SPLINE
SPL {X  -162.485, Y  +370.062, Z    +0.000, E1   +10.606, E3 +565885.380}
SPL {X  -162.818, Y  +379.636, Z    +0.000, E1    +5.115, E3 +565874.729}
SPL {X  -162.820, Y  +386.976, Z    +0.000, E1    +0.144, E3 +565873.828}
SPL {X  -162.820, Y  +391.982, Z    +0.000, E1    -3.443, E3 +565880.593}
SPL {X  -162.820, Y  +399.630, Z    +0.000, E1    -9.426, E3 +565883.100}
SPL {X  -162.820, Y  +408.127, Z    +0.000, E1   -18.417, E3 +565869.388}
SPL {X  -162.820, Y  +420.083, Z    +0.000, E1   -24.325, E3 +565889.864}
SPL {X  -162.820, Y  +428.527, Z    +0.000, E1   -26.988, E3 +565907.156}
SPL {X  -162.820, Y  +431.336, Z    +0.000, E1   -24.162, E3 +565937.366}
SPL {X  -162.820, Y  +432.048, Z    +0.000, E1   -22.832, E3 +565951.870}
SPL {X  -162.820, Y  +434.888, Z    +0.000, E1   -22.823, E3 +565965.819}
SPL {X  -162.820, Y  +436.834, Z    +0.000, E1   -22.779, E3 +565975.779}
SPL {X  -162.820, Y  +438.868, Z    +0.000, E1   -22.837, E3 +565985.433}
SPL {X  -162.820, Y  +441.351, Z    +0.000, E1   -22.805, E3 +565998.008}
SPL {X  -162.820, Y  +443.809, Z    +0.000, E1   -22.804, E3 +566010.174}
SPL {X  -162.820, Y  +446.105, Z    +0.000, E1   -22.815, E3 +566021.417}
SPL {X  -162.820, Y  +447.974, Z    +0.000, E1   -22.856, E3 +566030.320}
SPL {X  -162.820, Y  +449.911, Z    +0.000, E1   -22.774, E3 +566040.594}
SPL {X  -162.820, Y  +451.861, Z    +0.000, E1   -22.750, E3 +566050.442}
SPL {X  -162.820, Y  +454.167, Z    +0.000, E1   -22.842, E3 +566061.171}
SPL {X  -162.820, Y  +456.529, Z    +0.000, E1   -22.855, E3 +566072.700}
SPL {X  -162.820, Y  +458.725, Z    +0.000, E1   -22.793, E3 +566084.104}
SPL {X  -162.820, Y  +460.754, Z    +0.000, E1   -22.806, E3 +566093.977}
SPL {X  -162.820, Y  +462.409, Z    +0.000, E1   -22.783, E3 +566102.394}
SPL {X  -162.820, Y  +464.633, Z    +0.000, E1   -22.813, E3 +566113.223}
SPL {X  -162.820, Y  +467.913, Z    +0.000, E1   -22.879, E3 +566129.062}
SPL {X  -162.820, Y  +470.892, Z    +0.000, E1   -22.837, E3 +566143.952}
SPL {X  -162.820, Y  +472.726, Z    +0.000, E1   -22.777, E3 +566153.490}
SPL {X  -162.820, Y  +475.118, Z    +0.000, E1   -22.777, E3 +566165.462}
SPL {X  -162.820, Y  +478.177, Z    +0.000, E1   -22.834, E3 +566180.155}
SPL {X  -162.820, Y  +481.034, Z    +0.000, E1   -22.831, E3 +566194.292}
SPL {X  -162.820, Y  +483.391, Z    +0.000, E1   -22.793, E3 +566206.228}
SPL {X  -162.820, Y  +486.307, Z    +0.000, E1   -22.833, E3 +566220.482}
SPL {X  -162.820, Y  +488.828, Z    +0.000, E1   -22.793, E3 +566233.125}
SPL {X  -162.820, Y  +491.768, Z    +0.000, E1   -22.852, E3 +566247.422}
SPL {X  -162.820, Y  +495.526, Z    +0.000, E1   -22.833, E3 +566266.193}
SPL {X  -162.820, Y  +499.330, Z    +0.000, E1   -22.841, E3 +566284.974}
SPL {X  -162.820, Y  +503.049, Z    +0.000, E1   -22.823, E3 +566303.524}
SPL {X  -162.820, Y  +506.908, Z    +0.000, E1   -22.877, E3 +566322.194}
SPL {X  -162.820, Y  +510.068, Z    +0.000, E1   -22.761, E3 +566338.665}
SPL {X  -162.820, Y  +512.359, Z    +0.000, E1   -22.823, E3 +566349.397}
SPL {X  -162.820, Y  +513.873, Z    +0.000, E1   -22.800, E3 +566357.083}
SPL {X  -162.820, Y  +516.100, Z    +0.000, E1   -22.809, E3 +566368.160}
SPL {X  -162.820, Y  +518.662, Z    +0.000, E1   -22.847, E3 +566380.459}
SPL {X  -162.820, Y  +520.641, Z    +0.000, E1   -22.790, E3 +566390.699}
SPL {X  -162.820, Y  +523.535, Z    +0.000, E1   -22.857, E3 +566404.668}
SPL {X  -162.820, Y  +526.661, Z    +0.000, E1   -22.801, E3 +566420.492}
SPL {X  -162.820, Y  +528.725, Z    +0.000, E1   -22.770, E3 +566430.862}
SPL {X  -162.820, Y  +530.303, Z    +0.000, E1   -22.798, E3 +566438.481}
SPL {X  -162.820, Y  +532.614, Z    +0.000, E1   -22.828, E3 +566449.749}
SPL {X  -162.820, Y  +534.838, Z    +0.000, E1   -22.864, E3 +566460.378}
SPL {X  -162.820, Y  +536.882, Z    +0.000, E1   -22.782, E3 +566471.233}
SPL {X  -162.820, Y  +539.194, Z    +0.000, E1   -22.826, E3 +566482.282}
SPL {X  -162.820, Y  +541.555, Z    +0.000, E1   -22.817, E3 +566494.096}
SPL {X  -162.820, Y  +543.728, Z    +0.000, E1   -22.799, E3 +566504.954}
SPL {X  -162.820, Y  +545.925, Z    +0.000, E1   -22.803, E3 +566515.823}
SPL {X  -162.820, Y  +548.328, Z    +0.000, E1   -22.796, E3 +566527.819}
SPL {X  -162.820, Y  +551.027, Z    +0.000, E1   -22.819, E3 +566541.012}
SPL {X  -162.820, Y  +553.721, Z    +0.000, E1   -22.807, E3 +566554.456}
SPL {X  -162.820, Y  +556.430, Z    +0.000, E1   -22.821, E3 +566567.752}
SPL {X  -162.820, Y  +559.675, Z    +0.000, E1   -22.837, E3 +566583.832}
SPL {X  -162.820, Y  +562.799, Z    +0.000, E1   -22.814, E3 +566599.338}
SPL {X  -162.820, Y  +565.170, Z    +0.000, E1   -22.801, E3 +566611.163}
SPL {X  -162.820, Y  +568.020, Z    +0.000, E1   -22.787, E3 +566625.550}
SPL {X  -162.820, Y  +570.992, Z    +0.000, E1   -22.834, E3 +566639.769}
SPL {X  -162.820, Y  +572.901, Z    +0.000, E1   -22.775, E3 +566649.638}
SPL {X  -162.820, Y  +575.638, Z    +0.000, E1   -22.855, E3 +566662.747}
SPL {X  -162.820, Y  +578.553, Z    +0.000, E1   -22.801, E3 +566677.459}
SPL {X  -162.820, Y  +581.064, Z    +0.000, E1   -22.823, E3 +566689.744}
SPL {X  -162.820, Y  +583.435, Z    +0.000, E1   -22.808, E3 +566701.565}
SPL {X  -162.820, Y  +585.410, Z    +0.000, E1   -22.764, E3 +566711.701}
SPL {X  -162.820, Y  +587.676, Z    +0.000, E1   -22.853, E3 +566722.216}
SPL {X  -162.820, Y  +589.682, Z    +0.000, E1   -22.776, E3 +566732.746}
SPL {X  -162.820, Y  +591.720, Z    +0.000, E1   -22.868, E3 +566742.057}
SPL {X  -162.820, Y  +593.650, Z    +0.000, E1   -22.810, E3 +566752.126}
SPL {X  -162.820, Y  +595.830, Z    +0.000, E1   -22.828, E3 +566762.742}
SPL {X  -162.820, Y  +598.094, Z    +0.000, E1   -22.843, E3 +566773.855}
SPL {X  -162.820, Y  +600.420, Z    +0.000, E1   -22.826, E3 +566785.487}
SPL {X  -162.820, Y  +602.573, Z    +0.000, E1   -22.830, E3 +566796.072}
SPL {X  -162.820, Y  +604.828, Z    +0.000, E1   -22.784, E3 +566807.710}
SPL {X  -162.820, Y  +608.133, Z    +0.000, E1   -22.831, E3 +566823.828}
SPL {X  -162.820, Y  +611.103, Z    +0.000, E1   -22.785, E3 +566838.754}
SPL {X  -162.820, Y  +613.294, Z    +0.000, E1   -22.780, E3 +566849.627}
SPL {X  -162.820, Y  +615.356, Z    +0.000, E1   -22.799, E3 +566859.684}
SPL {X  -162.820, Y  +617.439, Z    +0.000, E1   -22.808, E3 +566869.942}
SPL {X  -162.820, Y  +619.665, Z    +0.000, E1   -22.817, E3 +566880.910}
SPL {X  -162.820, Y  +621.733, Z    +0.000, E1   -22.759, E3 +566891.634}
SPL {X  -162.820, Y  +624.076, Z    +0.000, E1   -22.774, E3 +566903.139}
SPL {X  -162.820, Y  +627.244, Z    +0.000, E1   -22.803, E3 +566918.822}
SPL {X  -162.820, Y  +630.349, Z    +0.000, E1   -22.766, E3 +566934.354}
SPL {X  -162.820, Y  +632.572, Z    +0.000, E1   -22.785, E3 +566945.160}
SPL {X  -162.820, Y  +634.507, Z    +0.000, E1   -22.784, E3 +566954.799}
SPL {X  -162.820, Y  +636.863, Z    +0.000, E1   -22.760, E3 +566966.721}
SPL {X  -162.820, Y  +640.111, Z    +0.000, E1   -22.809, E3 +566982.604}
SPL {X  -162.820, Y  +643.449, Z    +0.000, E1   -22.796, E3 +566999.122}
SPL {X  -162.820, Y  +645.630, Z    +0.000, E1   -22.795, E3 +567009.818}
SPL {X  -162.820, Y  +647.561, Z    +0.000, E1   -22.705, E3 +567020.268}
SPL {X  -162.820, Y  +651.051, Z    +0.000, E1   -22.833, E3 +567036.688}
SPL {X  -162.820, Y  +653.898, Z    +0.000, E1   -22.796, E3 +567050.874}
SPL {X  -162.820, Y  +656.161, Z    +0.000, E1   -22.812, E3 +567061.995}
SPL {X  -162.820, Y  +658.384, Z    +0.000, E1   -22.822, E3 +567072.862}
SPL {X  -162.820, Y  +660.215, Z    +0.000, E1   -22.649, E3 +567083.452}
SPL {X  -162.820, Y  +662.823, Z    +0.000, E1   -22.799, E3 +567095.160}
SPL {X  -162.820, Y  +665.862, Z    +0.000, E1   -22.864, E3 +567109.860}
SPL {X  -162.820, Y  +668.960, Z    +0.000, E1   -22.773, E3 +567125.810}
SPL {X  -162.820, Y  +671.605, Z    +0.000, E1   -22.777, E3 +567138.884}
SPL {X  -162.817, Y  +674.515, Z    +0.000, E1   -22.816, E3 +567153.081}
SPL {X  -162.773, Y  +677.428, Z    +0.000, E1   -22.762, E3 +567167.889}
SPL {X  -162.691, Y  +679.987, Z    +0.000, E1   -22.794, E3 +567180.302}
SPL {X  -162.559, Y  +682.717, Z    +0.000, E1   -22.726, E3 +567194.486}
SPL {X  -162.404, Y  +685.137, Z    +0.000, E1   -22.766, E3 +567206.008}
SPL {X  -162.229, Y  +687.364, Z    +0.000, E1   -22.685, E3 +567217.876}
SPL {X  -161.938, Y  +690.422, Z    +0.000, E1   -22.769, E3 +567232.283}
SPL {X  -161.065, Y  +697.344, Z    +0.000, E1   -25.698, E3 +567241.402}
SPL {X  -158.730, Y  +709.763, Z    +0.000, E1   -31.225, E3 +567250.075}
ENDSPLINE

SPLINE
SPL {X  -160.932, Y  +698.225, Z    +0.000, E1   -21.712, E3 +567281.185}
SPL {X  -161.691, Y  +692.643, Z    +0.000, E1   -17.369, E3 +567298.068}
SPL {X  -162.534, Y  +683.153, Z    +0.000, E1   -10.475, E3 +567323.535}
SPL {X  -162.820, Y  +667.630, Z    +0.000, E1    -0.882, E3 +567317.511}
SPL {X  -162.820, Y  +661.883, Z    +0.000, E1    +3.373, E3 +567322.954}
SPL {X  -162.820, Y  +655.163, Z    +0.000, E1    +8.702, E3 +567322.553}
SPL {X  -162.820, Y  +634.515, Z    +0.000, E1   +26.439, E3 +567314.966}
ENDSPLINE

SPLINE
SPL {X  -162.820, Y  +638.080, Z    +0.000, E1   +18.858, E3 +567344.931}
ENDSPLINE

SPLINE
SPL {X  -162.820, Y  +623.278, Z    +0.000, E1   +28.723, E3 +567346.501}
SPL {X  -162.820, Y  +618.658, Z    +0.000, E1   +26.841, E3 +567375.110}
ENDSPLINE

SPLINE
SPL {X  -162.820, Y  +623.685, Z    +0.000, E1   +22.346, E3 +567387.417}
ENDSPLINE

SPLINE
SPL {X  -162.820, Y  +621.304, Z    +0.000, E1   +22.259, E3 +567400.232}
SPL {X  -162.820, Y  +618.758, Z    +0.000, E1   +22.239, E3 +567413.383}
SPL {X  -162.820, Y  +616.062, Z    +0.000, E1   +22.275, E3 +567426.803}
SPL {X  -162.820, Y  +613.536, Z    +0.000, E1   +22.242, E3 +567439.925}
SPL {X  -162.820, Y  +611.128, Z    +0.000, E1   +22.252, E3 +567452.096}
SPL {X  -162.820, Y  +608.428, Z    +0.000, E1   +22.255, E3 +567465.879}
SPL {X  -162.820, Y  +605.984, Z    +0.000, E1   +22.221, E3 +567478.516}
SPL {X  -162.820, Y  +603.020, Z    +0.000, E1   +22.272, E3 +567493.414}
SPL {X  -162.820, Y  +599.168, Z    +0.000, E1   +22.310, E3 +567512.682}
SPL {X  -162.820, Y  +595.597, Z    +0.000, E1   +22.284, E3 +567531.018}
SPL {X  -162.820, Y  +593.320, Z    +0.000, E1   +22.199, E3 +567543.109}
SPL {X  -162.820, Y  +591.031, Z    +0.000, E1   +22.283, E3 +567554.200}
SPL {X  -162.820, Y  +588.026, Z    +0.000, E1   +22.301, E3 +567569.327}
SPL {X  -162.820, Y  +585.899, Z    +0.000, E1   +22.286, E3 +567580.129}
SPL {X  -162.820, Y  +583.204, Z    +0.000, E1   +22.278, E3 +567594.152}
SPL {X  -162.820, Y  +579.691, Z    +0.000, E1   +22.312, E3 +567611.639}
SPL {X  -162.820, Y  +577.460, Z    +0.000, E1   +22.218, E3 +567623.627}
SPL {X  -162.820, Y  +575.394, Z    +0.000, E1   +22.240, E3 +567634.052}
SPL {X  -162.820, Y  +572.645, Z    +0.000, E1   +22.246, E3 +567648.049}
SPL {X  -162.820, Y  +570.282, Z    +0.000, E1   +22.231, E3 +567660.100}
SPL {X  -162.820, Y  +567.961, Z    +0.000, E1   +22.247, E3 +567671.889}
SPL {X  -162.820, Y  +564.506, Z    +0.000, E1   +22.298, E3 +567689.203}
SPL {X  -162.820, Y  +561.620, Z    +0.000, E1   +22.191, E3 +567704.584}
SPL {X  -162.820, Y  +559.515, Z    +0.000, E1   +22.273, E3 +567714.586}
SPL {X  -162.820, Y  +556.723, Z    +0.000, E1   +22.309, E3 +567728.670}
SPL {X  -162.820, Y  +554.378, Z    +0.000, E1   +22.288, E3 +567740.515}
SPL {X  -162.820, Y  +552.787, Z    +0.000, E1   +22.213, E3 +567749.337}
SPL {X  -162.820, Y  +550.871, Z    +0.000, E1   +22.229, E3 +567758.932}
SPL {X  -162.820, Y  +548.168, Z    +0.000, E1   +22.298, E3 +567772.268}
SPL {X  -162.820, Y  +545.860, Z    +0.000, E1   +22.216, E3 +567784.525}
SPL {X  -162.820, Y  +543.558, Z    +0.000, E1   +22.285, E3 +567795.756}
SPL {X  -162.820, Y  +540.968, Z    +0.000, E1   +22.274, E3 +567809.028}
SPL {X  -162.820, Y  +537.857, Z    +0.000, E1   +22.280, E3 +567824.904}
SPL {X  -162.820, Y  +534.880, Z    +0.000, E1   +22.252, E3 +567840.172}
SPL {X  -162.820, Y  +532.896, Z    +0.000, E1   +22.234, E3 +567850.333}
SPL {X  -162.820, Y  +531.056, Z    +0.000, E1   +22.251, E3 +567859.615}
SPL {X  -162.820, Y  +528.708, Z    +0.000, E1   +22.319, E3 +567870.996}
SPL {X  -162.820, Y  +525.932, Z    +0.000, E1   +22.258, E3 +567885.753}
SPL {X  -162.820, Y  +522.524, Z    +0.000, E1   +22.326, E3 +567902.476}
SPL {X  -162.820, Y  +519.457, Z    +0.000, E1   +22.481, E3 +567916.605}
SPL {X  -162.820, Y  +506.285, Z    +0.000, E1   +28.538, E3 +567928.063}
SPL {X  -162.820, Y  +504.441, Z    +0.000, E1   +27.574, E3 +567942.406}
SPL {X  -162.820, Y  +502.813, Z    +0.000, E1   +26.013, E3 +567960.603}
SPL {X  -162.820, Y  +502.016, Z    +0.000, E1   +24.802, E3 +567972.946}
SPL {X  -162.820, Y  +501.060, Z    +0.000, E1   +24.081, E3 +567983.135}
SPL {X  -162.820, Y  +499.934, Z    +0.000, E1   +22.814, E3 +567999.004}
SPL {X  -162.820, Y  +498.303, Z    +0.000, E1   +21.749, E3 +568016.260}
SPL {X  -162.820, Y  +495.897, Z    +0.000, E1   +21.662, E3 +568029.414}
SPL {X  -162.820, Y  +493.717, Z    +0.000, E1   +21.704, E3 +568040.520}
SPL {X  -162.820, Y  +491.396, Z    +0.000, E1   +21.707, E3 +568052.644}
SPL {X  -162.820, Y  +489.485, Z    +0.000, E1   +21.661, E3 +568062.992}
SPL {X  -162.820, Y  +487.723, Z    +0.000, E1   +21.665, E3 +568072.195}
SPL {X  -162.820, Y  +485.661, Z    +0.000, E1   +21.712, E3 +568082.639}
SPL {X  -162.820, Y  +482.775, Z    +0.000, E1   +21.716, E3 +568097.891}
SPL {X  -162.820, Y  +479.894, Z    +0.000, E1   +21.695, E3 +568112.967}
SPL {X  -162.820, Y  +477.685, Z    +0.000, E1   +21.656, E3 +568124.905}
SPL {X  -162.820, Y  +475.419, Z    +0.000, E1   +21.711, E3 +568136.258}
SPL {X  -162.820, Y  +473.301, Z    +0.000, E1   +21.712, E3 +568147.355}
SPL {X  -162.820, Y  +470.965, Z    +0.000, E1   +21.700, E3 +568159.700}
SPL {X  -162.820, Y  +469.036, Z    +0.000, E1   +21.695, E3 +568169.743}
SPL {X  -162.820, Y  +467.138, Z    +0.000, E1   +21.678, E3 +568179.915}
SPL {X  -162.820, Y  +465.011, Z    +0.000, E1   +21.692, E3 +568190.898}
SPL {X  -162.820, Y  +462.669, Z    +0.000, E1   +21.752, E3 +568202.678}
SPL {X  -162.820, Y  +460.725, Z    +0.000, E1   +21.689, E3 +568213.291}
SPL {X  -162.820, Y  +458.666, Z    +0.000, E1   +21.695, E3 +568224.103}
SPL {X  -162.820, Y  +456.431, Z    +0.000, E1   +21.708, E3 +568235.632}
SPL {X  -162.820, Y  +454.628, Z    +0.000, E1   +21.674, E3 +568245.350}
SPL {X  -162.820, Y  +452.690, Z    +0.000, E1   +21.773, E3 +568254.624}
SPL {X  -162.820, Y  +450.610, Z    +0.000, E1   +21.698, E3 +568266.223}
SPL {X  -162.820, Y  +448.170, Z    +0.000, E1   +21.667, E3 +568279.244}
SPL {X  -162.820, Y  +446.246, Z    +0.000, E1   +21.696, E3 +568289.061}
SPL {X  -162.820, Y  +443.784, Z    +0.000, E1   +21.713, E3 +568301.848}
SPL {X  -162.820, Y  +440.567, Z    +0.000, E1   +21.731, E3 +568318.687}
SPL {X  -162.820, Y  +437.628, Z    +0.000, E1   +21.678, E3 +568334.351}
SPL {X  -162.820, Y  +435.262, Z    +0.000, E1   +21.727, E3 +568346.287}
SPL {X  -162.820, Y  +433.510, Z    +0.000, E1   +21.692, E3 +568355.701}
SPL {X  -162.820, Y  +431.492, Z    +0.000, E1   +21.686, E3 +568366.396}
SPL {X  -162.820, Y  +429.074, Z    +0.000, E1   +21.710, E3 +568378.848}
SPL {X  -162.820, Y  +427.020, Z    +0.000, E1   +21.674, E3 +568389.850}
SPL {X  -162.820, Y  +424.525, Z    +0.000, E1   +21.712, E3 +568402.763}
SPL {X  -162.820, Y  +421.144, Z    +0.000, E1   +21.719, E3 +568420.430}
SPL {X  -162.820, Y  +418.116, Z    +0.000, E1   +21.761, E3 +568435.761}
SPL {X  -162.820, Y  +416.127, Z    +0.000, E1   +21.715, E3 +568446.466}
SPL {X  -162.820, Y  +414.361, Z    +0.000, E1   +21.613, E3 +568456.653}
SPL {X  -162.820, Y  +411.450, Z    +0.000, E1   +21.710, E3 +568471.227}
SPL {X  -162.820, Y  +408.590, Z    +0.000, E1   +21.735, E3 +568485.852}
SPL {X  -162.820, Y  +406.238, Z    +0.000, E1   +21.697, E3 +568498.501}
SPL {X  -162.820, Y  +403.166, Z    +0.000, E1   +21.746, E3 +568514.307}
SPL {X  -162.820, Y  +400.348, Z    +0.000, E1   +21.713, E3 +568529.142}
SPL {X  -162.820, Y  +398.298, Z    +0.000, E1   +21.721, E3 +568539.757}
SPL {X  -162.820, Y  +396.371, Z    +0.000, E1   +21.713, E3 +568549.939}
SPL {X  -162.820, Y  +394.508, Z    +0.000, E1   +21.616, E3 +568560.495}
SPL {X  -162.820, Y  +391.777, Z    +0.000, E1   +21.714, E3 +568574.154}
SPL {X  -162.820, Y  +388.822, Z    +0.000, E1   +21.717, E3 +568589.474}
SPL {X  -162.820, Y  +386.818, Z    +0.000, E1   +21.679, E3 +568600.214}
SPL {X  -162.820, Y  +384.697, Z    +0.000, E1   +21.693, E3 +568611.284}
SPL {X  -162.820, Y  +382.288, Z    +0.000, E1   +21.742, E3 +568623.407}
SPL {X  -162.817, Y  +379.520, Z    +0.000, E1   +21.723, E3 +568638.245}
SPL {X  -162.776, Y  +376.710, Z    +0.000, E1   +21.698, E3 +568652.984}
SPL {X  -162.707, Y  +374.438, Z    +0.000, E1   +21.688, E3 +568664.988}
SPL {X  -162.607, Y  +372.171, Z    +0.000, E1   +21.692, E3 +568676.788}
SPL {X  -162.494, Y  +370.197, Z    +0.000, E1   +21.655, E3 +568687.414}
SPL {X  -162.349, Y  +368.131, Z    +0.000, E1   +21.624, E3 +568698.532}
SPL {X  -162.161, Y  +365.866, Z    +0.000, E1   +21.642, E3 +568710.217}
SPL {X  -161.651, Y  +361.024, Z    +0.000, E1   +22.970, E3 +568723.640}
SPL {X  -160.281, Y  +351.857, Z    +0.000, E1   +24.243, E3 +568758.979}
ENDSPLINE

SPLINE
SPL {X  -161.833, Y  +362.603, Z    +0.000, E1   +17.021, E3 +568773.675}
ENDSPLINE

SPLINE
SPL {X  -160.786, Y  +354.842, Z    +0.000, E1   +19.274, E3 +568805.831}
ENDSPLINE

SPLINE
SPL {X  -162.485, Y  +370.062, Z    +0.000, E1   +10.606, E3 +568812.209}
SPL {X  -162.818, Y  +379.636, Z    +0.000, E1    +5.115, E3 +568801.558}
SPL {X  -162.820, Y  +386.976, Z    +0.000, E1    +0.144, E3 +568800.657}
SPL {X  -162.820, Y  +391.982, Z    +0.000, E1    -3.443, E3 +568807.422}
SPL {X  -162.820, Y  +399.630, Z    +0.000, E1    -9.426, E3 +568809.929}
SPL {X  -162.820, Y  +408.127, Z    +0.000, E1   -18.417, E3 +568796.218}
SPL {X  -162.820, Y  +420.083, Z    +0.000, E1   -24.325, E3 +568816.693}
SPL {X  -162.820, Y  +428.527, Z    +0.000, E1   -26.988, E3 +568833.985}
SPL {X  -162.820, Y  +431.336, Z    +0.000, E1   -24.162, E3 +568864.195}
SPL {X  -162.820, Y  +432.048, Z    +0.000, E1   -22.832, E3 +568878.699}
SPL {X  -162.820, Y  +434.888, Z    +0.000, E1   -22.823, E3 +568892.648}
SPL {X  -162.820, Y  +436.834, Z    +0.000, E1   -22.779, E3 +568902.609}
SPL {X  -162.820, Y  +438.868, Z    +0.000, E1   -22.837, E3 +568912.262}
SPL {X  -162.820, Y  +441.351, Z    +0.000, E1   -22.805, E3 +568924.837}
SPL {X  -162.820, Y  +443.809, Z    +0.000, E1   -22.804, E3 +568937.004}
SPL {X  -162.820, Y  +446.105, Z    +0.000, E1   -22.815, E3 +568948.246}
SPL {X  -162.820, Y  +447.974, Z    +0.000, E1   -22.856, E3 +568957.149}
SPL {X  -162.820, Y  +449.911, Z    +0.000, E1   -22.774, E3 +568967.424}
SPL {X  -162.820, Y  +451.861, Z    +0.000, E1   -22.750, E3 +568977.271}
SPL {X  -162.820, Y  +454.167, Z    +0.000, E1   -22.842, E3 +568988.001}
SPL {X  -162.820, Y  +456.529, Z    +0.000, E1   -22.855, E3 +568999.529}
SPL {X  -162.820, Y  +458.725, Z    +0.000, E1   -22.793, E3 +569010.933}
SPL {X  -162.820, Y  +460.754, Z    +0.000, E1   -22.806, E3 +569020.806}
SPL {X  -162.820, Y  +462.409, Z    +0.000, E1   -22.783, E3 +569029.223}
SPL {X  -162.820, Y  +464.633, Z    +0.000, E1   -22.813, E3 +569040.053}
SPL {X  -162.820, Y  +467.913, Z    +0.000, E1   -22.879, E3 +569055.892}
SPL {X  -162.820, Y  +470.892, Z    +0.000, E1   -22.837, E3 +569070.781}
SPL {X  -162.820, Y  +472.726, Z    +0.000, E1   -22.777, E3 +569080.320}
SPL {X  -162.820, Y  +475.118, Z    +0.000, E1   -22.777, E3 +569092.291}
SPL {X  -162.820, Y  +477.389, Z    +0.000, E1   -22.803, E3 +569103.208}
SPL {X  -162.820, Y  +478.914, Z    +0.000, E1   -22.821, E3 +569110.599}
SPL {X  -162.820, Y  +481.034, Z    +0.000, E1   -22.831, E3 +569121.122}
SPL {X  -162.820, Y  +484.256, Z    +0.000, E1   -22.840, E3 +569137.140}
SPL {X  -162.820, Y  +487.952, Z    +0.000, E1   -22.824, E3 +569155.570}
SPL {X  -162.820, Y  +490.653, Z    +0.000, E1   -22.810, E3 +569168.840}
SPL {X  -162.820, Y  +493.233, Z    +0.000, E1   -22.844, E3 +569181.518}
SPL {X  -162.820, Y  +496.150, Z    +0.000, E1   -22.796, E3 +569196.238}
SPL {X  -162.820, Y  +498.661, Z    +0.000, E1   -22.828, E3 +569208.419}
SPL {X  -162.820, Y  +501.761, Z    +0.000, E1   -22.820, E3 +569223.987}
SPL {X  -162.820, Y  +505.323, Z    +0.000, E1   -22.838, E3 +569241.434}
SPL {X  -162.820, Y  +507.875, Z    +0.000, E1   -22.849, E3 +569253.801}
SPL {X  -162.820, Y  +510.068, Z    +0.000, E1   -22.761, E3 +569265.495}
SPL {X  -162.820, Y  +512.359, Z    +0.000, E1   -22.823, E3 +569276.226}
SPL {X  -162.820, Y  +514.562, Z    +0.000, E1   -22.806, E3 +569287.413}
SPL {X  -162.820, Y  +517.952, Z    +0.000, E1   -22.864, E3 +569303.810}
SPL {X  -162.820, Y  +520.641, Z    +0.000, E1   -22.790, E3 +569317.529}
SPL {X  -162.820, Y  +522.740, Z    +0.000, E1   -22.811, E3 +569327.771}
SPL {X  -162.820, Y  +524.628, Z    +0.000, E1   -22.846, E3 +569336.766}
SPL {X  -162.820, Y  +526.661, Z    +0.000, E1   -22.801, E3 +569347.322}
SPL {X  -162.820, Y  +529.662, Z    +0.000, E1   -22.810, E3 +569362.172}
SPL {X  -162.820, Y  +532.614, Z    +0.000, E1   -22.828, E3 +569376.579}
SPL {X  -162.820, Y  +534.838, Z    +0.000, E1   -22.864, E3 +569387.208}
SPL {X  -162.820, Y  +536.882, Z    +0.000, E1   -22.782, E3 +569398.063}
SPL {X  -162.820, Y  +539.194, Z    +0.000, E1   -22.826, E3 +569409.111}
SPL {X  -162.820, Y  +541.555, Z    +0.000, E1   -22.817, E3 +569420.925}
SPL {X  -162.820, Y  +543.728, Z    +0.000, E1   -22.799, E3 +569431.783}
SPL {X  -162.820, Y  +545.925, Z    +0.000, E1   -22.803, E3 +569442.653}
SPL {X  -162.820, Y  +548.328, Z    +0.000, E1   -22.796, E3 +569454.648}
SPL {X  -162.820, Y  +551.027, Z    +0.000, E1   -22.819, E3 +569467.841}
SPL {X  -162.820, Y  +553.721, Z    +0.000, E1   -22.807, E3 +569481.285}
SPL {X  -162.820, Y  +556.430, Z    +0.000, E1   -22.821, E3 +569494.581}
SPL {X  -162.820, Y  +558.974, Z    +0.000, E1   -22.806, E3 +569507.281}
SPL {X  -162.820, Y  +562.171, Z    +0.000, E1   -22.845, E3 +569522.979}
SPL {X  -162.820, Y  +565.170, Z    +0.000, E1   -22.801, E3 +569537.993}
SPL {X  -162.820, Y  +567.308, Z    +0.000, E1   -22.750, E3 +569549.009}
SPL {X  -162.820, Y  +570.378, Z    +0.000, E1   -22.843, E3 +569563.633}
SPL {X  -162.820, Y  +573.634, Z    +0.000, E1   -22.827, E3 +569579.776}
SPL {X  -162.820, Y  +576.228, Z    +0.000, E1   -22.814, E3 +569592.673}
SPL {X  -162.820, Y  +578.553, Z    +0.000, E1   -22.801, E3 +569604.289}
SPL {X  -162.820, Y  +581.064, Z    +0.000, E1   -22.823, E3 +569616.573}
SPL {X  -162.820, Y  +583.435, Z    +0.000, E1   -22.808, E3 +569628.395}
SPL {X  -162.820, Y  +585.410, Z    +0.000, E1   -22.764, E3 +569638.530}
SPL {X  -162.820, Y  +587.676, Z    +0.000, E1   -22.853, E3 +569649.045}
SPL {X  -162.820, Y  +590.707, Z    +0.000, E1   -22.855, E3 +569664.195}
SPL {X  -162.820, Y  +593.650, Z    +0.000, E1   -22.810, E3 +569678.956}
SPL {X  -162.820, Y  +595.830, Z    +0.000, E1   -22.828, E3 +569689.571}
SPL {X  -162.820, Y  +598.094, Z    +0.000, E1   -22.843, E3 +569700.685}
SPL {X  -162.820, Y  +600.420, Z    +0.000, E1   -22.826, E3 +569712.316}
SPL {X  -162.820, Y  +602.573, Z    +0.000, E1   -22.830, E3 +569722.901}
SPL {X  -162.820, Y  +604.828, Z    +0.000, E1   -22.784, E3 +569734.539}
SPL {X  -162.820, Y  +608.133, Z    +0.000, E1   -22.831, E3 +569750.657}
SPL {X  -162.820, Y  +611.103, Z    +0.000, E1   -22.785, E3 +569765.583}
SPL {X  -162.820, Y  +613.294, Z    +0.000, E1   -22.780, E3 +569776.456}
SPL {X  -162.820, Y  +615.356, Z    +0.000, E1   -22.799, E3 +569786.513}
SPL {X  -162.820, Y  +617.439, Z    +0.000, E1   -22.808, E3 +569796.771}
SPL {X  -162.820, Y  +619.665, Z    +0.000, E1   -22.817, E3 +569807.739}
SPL {X  -162.820, Y  +621.733, Z    +0.000, E1   -22.759, E3 +569818.464}
SPL {X  -162.820, Y  +624.076, Z    +0.000, E1   -22.774, E3 +569829.969}
SPL {X  -162.820, Y  +627.244, Z    +0.000, E1   -22.803, E3 +569845.651}
SPL {X  -162.820, Y  +630.349, Z    +0.000, E1   -22.766, E3 +569861.183}
SPL {X  -162.820, Y  +632.572, Z    +0.000, E1   -22.785, E3 +569871.989}
SPL {X  -162.820, Y  +634.507, Z    +0.000, E1   -22.784, E3 +569881.628}
SPL {X  -162.820, Y  +636.863, Z    +0.000, E1   -22.760, E3 +569893.550}
SPL {X  -162.820, Y  +640.111, Z    +0.000, E1   -22.809, E3 +569909.433}
SPL {X  -162.820, Y  +643.449, Z    +0.000, E1   -22.796, E3 +569925.951}
SPL {X  -162.820, Y  +645.630, Z    +0.000, E1   -22.795, E3 +569936.647}
SPL {X  -162.820, Y  +647.561, Z    +0.000, E1   -22.705, E3 +569947.098}
SPL {X  -162.820, Y  +651.051, Z    +0.000, E1   -22.833, E3 +569963.517}
SPL {X  -162.820, Y  +653.898, Z    +0.000, E1   -22.796, E3 +569977.703}
SPL {X  -162.820, Y  +656.161, Z    +0.000, E1   -22.812, E3 +569988.825}
SPL {X  -162.820, Y  +658.384, Z    +0.000, E1   -22.822, E3 +569999.691}
SPL {X  -162.820, Y  +660.215, Z    +0.000, E1   -22.649, E3 +570010.281}
SPL {X  -162.820, Y  +662.823, Z    +0.000, E1   -22.799, E3 +570021.989}
SPL {X  -162.820, Y  +665.112, Z    +0.000, E1   -22.835, E3 +570033.044}
SPL {X  -162.820, Y  +667.016, Z    +0.000, E1   -22.823, E3 +570042.472}
SPL {X  -162.820, Y  +668.960, Z    +0.000, E1   -22.773, E3 +570052.640}
SPL {X  -162.820, Y  +672.333, Z    +0.000, E1   -22.837, E3 +570068.976}
SPL {X  -162.812, Y  +675.071, Z    +0.000, E1   -22.742, E3 +570083.121}
SPL {X  -162.773, Y  +677.428, Z    +0.000, E1   -22.762, E3 +570094.718}
SPL {X  -162.691, Y  +679.987, Z    +0.000, E1   -22.794, E3 +570107.132}
SPL {X  -162.559, Y  +682.717, Z    +0.000, E1   -22.726, E3 +570121.315}
SPL {X  -162.349, Y  +685.880, Z    +0.000, E1   -22.738, E3 +570136.916}
SPL {X  -162.164, Y  +688.106, Z    +0.000, E1   -22.661, E3 +570148.436}
SPL {X  -161.938, Y  +690.422, Z    +0.000, E1   -22.769, E3 +570159.112}
SPL {X  -161.065, Y  +697.344, Z    +0.000, E1   -25.698, E3 +570168.231}
SPL {X  -158.553, Y  +710.529, Z    +0.000, E1   -30.890, E3 +570182.128}
ENDSPLINE

SPLINE
SPL {X  -161.215, Y  +696.305, Z    +0.000, E1   -20.575, E3 +570208.709}
SPL {X  -161.691, Y  +692.643, Z    +0.000, E1   -17.369, E3 +570224.897}
SPL {X  -162.534, Y  +683.153, Z    +0.000, E1   -10.475, E3 +570250.364}
SPL {X  -162.820, Y  +667.630, Z    +0.000, E1    -0.882, E3 +570244.340}
SPL {X  -162.820, Y  +661.883, Z    +0.000, E1    +3.373, E3 +570249.784}
SPL {X  -162.820, Y  +653.808, Z    +0.000, E1    +9.891, E3 +570247.475}
SPL {X  -162.820, Y  +632.548, Z    +0.000, E1   +27.446, E3 +570244.011}
ENDSPLINE

SPLINE
SPL {X  -162.820, Y  +638.080, Z    +0.000, E1   +18.858, E3 +570271.760}
ENDSPLINE

SPLINE
SPL {X  -162.820, Y  +623.278, Z    +0.000, E1   +28.723, E3 +570273.331}
SPL {X  -162.820, Y  +618.658, Z    +0.000, E1   +26.841, E3 +570301.939}
ENDSPLINE

SPLINE
SPL {X  -162.820, Y  +623.685, Z    +0.000, E1   +22.346, E3 +570314.246}
ENDSPLINE

SPLINE
SPL {X  -162.820, Y  +621.304, Z    +0.000, E1   +22.259, E3 +570327.061}
SPL {X  -162.820, Y  +618.758, Z    +0.000, E1   +22.239, E3 +570340.212}
SPL {X  -162.820, Y  +616.062, Z    +0.000, E1   +22.275, E3 +570353.633}
SPL {X  -162.820, Y  +613.536, Z    +0.000, E1   +22.242, E3 +570366.754}
SPL {X  -162.820, Y  +611.128, Z    +0.000, E1   +22.252, E3 +570378.925}
SPL {X  -162.820, Y  +608.428, Z    +0.000, E1   +22.255, E3 +570392.708}
SPL {X  -162.820, Y  +605.178, Z    +0.000, E1   +22.267, E3 +570409.240}
SPL {X  -162.820, Y  +602.350, Z    +0.000, E1   +22.224, E3 +570423.858}
SPL {X  -162.820, Y  +599.842, Z    +0.000, E1   +22.298, E3 +570436.009}
SPL {X  -162.820, Y  +597.194, Z    +0.000, E1   +22.253, E3 +570449.930}
SPL {X  -162.820, Y  +594.779, Z    +0.000, E1   +22.284, E3 +570461.834}
SPL {X  -162.820, Y  +592.389, Z    +0.000, E1   +22.245, E3 +570474.451}
SPL {X  -162.820, Y  +589.492, Z    +0.000, E1   +22.304, E3 +570488.635}
SPL {X  -162.820, Y  +587.447, Z    +0.000, E1   +22.279, E3 +570499.164}
SPL {X  -162.820, Y  +585.192, Z    +0.000, E1   +22.298, E3 +570510.574}
SPL {X  -162.820, Y  +582.610, Z    +0.000, E1   +22.234, E3 +570524.198}
SPL {X  -162.820, Y  +580.317, Z    +0.000, E1   +22.300, E3 +570535.251}
SPL {X  -162.820, Y  +578.878, Z    +0.000, E1   +22.272, E3 +570542.761}
SPL {X  -162.820, Y  +576.856, Z    +0.000, E1   +22.233, E3 +570553.519}
SPL {X  -162.820, Y  +574.811, Z    +0.000, E1   +22.236, E3 +570563.783}
SPL {X  -162.820, Y  +572.645, Z    +0.000, E1   +22.246, E3 +570574.878}
SPL {X  -162.820, Y  +569.475, Z    +0.000, E1   +22.269, E3 +570590.885}
SPL {X  -162.820, Y  +565.838, Z    +0.000, E1   +22.271, E3 +570609.479}
SPL {X  -162.820, Y  +562.162, Z    +0.000, E1   +22.252, E3 +570628.296}
SPL {X  -162.820, Y  +558.919, Z    +0.000, E1   +22.286, E3 +570644.460}
SPL {X  -162.820, Y  +556.169, Z    +0.000, E1   +22.295, E3 +570658.289}
SPL {X  -162.820, Y  +553.294, Z    +0.000, E1   +22.266, E3 +570673.287}
SPL {X  -162.820, Y  +550.136, Z    +0.000, E1   +22.258, E3 +570689.400}
SPL {X  -162.820, Y  +546.694, Z    +0.000, E1   +22.290, E3 +570706.722}
SPL {X  -162.820, Y  +543.558, Z    +0.000, E1   +22.285, E3 +570722.585}
SPL {X  -162.820, Y  +541.633, Z    +0.000, E1   +22.257, E3 +570732.513}
SPL {X  -162.820, Y  +539.116, Z    +0.000, E1   +22.302, E3 +570745.124}
SPL {X  -162.820, Y  +536.913, Z    +0.000, E1   +22.192, E3 +570757.048}
SPL {X  -162.820, Y  +534.880, Z    +0.000, E1   +22.252, E3 +570767.002}
SPL {X  -162.820, Y  +532.896, Z    +0.000, E1   +22.234, E3 +570777.162}
SPL {X  -162.820, Y  +531.056, Z    +0.000, E1   +22.251, E3 +570786.444}
SPL {X  -162.820, Y  +528.708, Z    +0.000, E1   +22.319, E3 +570797.826}
SPL {X  -162.820, Y  +525.932, Z    +0.000, E1   +22.258, E3 +570812.582}
SPL {X  -162.820, Y  +522.524, Z    +0.000, E1   +22.326, E3 +570829.306}
SPL {X  -162.820, Y  +519.457, Z    +0.000, E1   +22.481, E3 +570843.435}
SPL {X  -162.820, Y  +506.285, Z    +0.000, E1   +28.538, E3 +570854.893}
SPL {X  -162.820, Y  +504.441, Z    +0.000, E1   +27.574, E3 +570869.235}
SPL {X  -162.820, Y  +503.215, Z    +0.000, E1   +26.369, E3 +570882.742}
SPL {X  -162.820, Y  +502.265, Z    +0.000, E1   +25.287, E3 +570895.224}
SPL {X  -162.820, Y  +501.060, Z    +0.000, E1   +24.081, E3 +570909.964}
SPL {X  -162.820, Y  +500.336, Z    +0.000, E1   +23.110, E3 +570921.104}
SPL {X  -162.820, Y  +499.240, Z    +0.000, E1   +22.316, E3 +570933.415}
SPL {X  -162.820, Y  +498.027, Z    +0.000, E1   +21.516, E3 +570946.323}
SPL {X  -162.820, Y  +495.897, Z    +0.000, E1   +21.662, E3 +570956.243}
SPL {X  -162.820, Y  +493.717, Z    +0.000, E1   +21.704, E3 +570967.349}
SPL {X  -162.820, Y  +491.396, Z    +0.000, E1   +21.707, E3 +570979.473}
SPL {X  -162.820, Y  +488.560, Z    +0.000, E1   +21.695, E3 +570994.583}
SPL {X  -162.820, Y  +485.661, Z    +0.000, E1   +21.712, E3 +571009.468}
SPL {X  -162.820, Y  +483.668, Z    +0.000, E1   +21.664, E3 +571020.296}
SPL {X  -162.820, Y  +481.739, Z    +0.000, E1   +21.704, E3 +571030.009}
SPL {X  -162.820, Y  +479.894, Z    +0.000, E1   +21.695, E3 +571039.797}
SPL {X  -162.820, Y  +477.685, Z    +0.000, E1   +21.656, E3 +571051.734}
SPL {X  -162.820, Y  +475.419, Z    +0.000, E1   +21.711, E3 +571063.087}
SPL {X  -162.820, Y  +473.301, Z    +0.000, E1   +21.712, E3 +571074.184}
SPL {X  -162.820, Y  +470.965, Z    +0.000, E1   +21.700, E3 +571086.529}
SPL {X  -162.820, Y  +469.036, Z    +0.000, E1   +21.695, E3 +571096.573}
SPL {X  -162.820, Y  +467.138, Z    +0.000, E1   +21.678, E3 +571106.744}
SPL {X  -162.820, Y  +465.011, Z    +0.000, E1   +21.692, E3 +571117.727}
SPL {X  -162.820, Y  +462.669, Z    +0.000, E1   +21.752, E3 +571129.507}
SPL {X  -162.820, Y  +460.725, Z    +0.000, E1   +21.689, E3 +571140.120}
SPL {X  -162.820, Y  +458.666, Z    +0.000, E1   +21.695, E3 +571150.932}
SPL {X  -162.820, Y  +456.431, Z    +0.000, E1   +21.708, E3 +571162.461}
SPL {X  -162.820, Y  +454.628, Z    +0.000, E1   +21.674, E3 +571172.179}
SPL {X  -162.820, Y  +452.690, Z    +0.000, E1   +21.773, E3 +571181.453}
SPL {X  -162.820, Y  +450.610, Z    +0.000, E1   +21.698, E3 +571193.052}
SPL {X  -162.820, Y  +448.170, Z    +0.000, E1   +21.667, E3 +571206.073}
SPL {X  -162.820, Y  +446.246, Z    +0.000, E1   +21.696, E3 +571215.891}
SPL {X  -162.820, Y  +443.784, Z    +0.000, E1   +21.713, E3 +571228.677}
SPL {X  -162.820, Y  +441.754, Z    +0.000, E1   +21.708, E3 +571239.229}
SPL {X  -162.820, Y  +439.933, Z    +0.000, E1   +21.690, E3 +571248.993}
SPL {X  -162.820, Y  +437.628, Z    +0.000, E1   +21.678, E3 +571261.181}
SPL {X  -162.820, Y  +435.262, Z    +0.000, E1   +21.727, E3 +571273.116}
SPL {X  -162.820, Y  +433.510, Z    +0.000, E1   +21.692, E3 +571282.530}
SPL {X  -162.820, Y  +431.492, Z    +0.000, E1   +21.686, E3 +571293.226}
SPL {X  -162.820, Y  +429.074, Z    +0.000, E1   +21.710, E3 +571305.677}
SPL {X  -162.820, Y  +427.020, Z    +0.000, E1   +21.674, E3 +571316.679}
SPL {X  -162.820, Y  +425.215, Z    +0.000, E1   +21.693, E3 +571325.981}
SPL {X  -162.820, Y  +422.986, Z    +0.000, E1   +21.685, E3 +571337.793}
SPL {X  -162.820, Y  +420.528, Z    +0.000, E1   +21.706, E3 +571350.443}
SPL {X  -162.820, Y  +418.116, Z    +0.000, E1   +21.761, E3 +571362.590}
SPL {X  -162.820, Y  +416.127, Z    +0.000, E1   +21.715, E3 +571373.295}
SPL {X  -162.820, Y  +414.361, Z    +0.000, E1   +21.613, E3 +571383.482}
SPL {X  -162.820, Y  +411.450, Z    +0.000, E1   +21.710, E3 +571398.056}
SPL {X  -162.820, Y  +408.590, Z    +0.000, E1   +21.735, E3 +571412.681}
SPL {X  -162.820, Y  +406.238, Z    +0.000, E1   +21.697, E3 +571425.330}
SPL {X  -162.820, Y  +404.001, Z    +0.000, E1   +21.723, E3 +571436.760}
SPL {X  -162.820, Y  +402.223, Z    +0.000, E1   +21.697, E3 +571446.245}
SPL {X  -162.820, Y  +400.348, Z    +0.000, E1   +21.713, E3 +571455.971}
SPL {X  -162.820, Y  +398.298, Z    +0.000, E1   +21.721, E3 +571466.587}
SPL {X  -162.820, Y  +396.371, Z    +0.000, E1   +21.713, E3 +571476.768}
SPL {X  -162.820, Y  +394.508, Z    +0.000, E1   +21.616, E3 +571487.324}
SPL {X  -162.820, Y  +392.435, Z    +0.000, E1   +21.681, E3 +571497.677}
SPL {X  -162.820, Y  +389.390, Z    +0.000, E1   +21.742, E3 +571513.284}
SPL {X  -162.820, Y  +386.818, Z    +0.000, E1   +21.679, E3 +571527.043}
SPL {X  -162.820, Y  +384.697, Z    +0.000, E1   +21.693, E3 +571538.113}
SPL {X  -162.820, Y  +382.288, Z    +0.000, E1   +21.742, E3 +571550.237}
SPL {X  -162.820, Y  +380.381, Z    +0.000, E1   +21.655, E3 +571560.962}
SPL {X  -162.808, Y  +378.512, Z    +0.000, E1   +21.736, E3 +571570.014}
SPL {X  -162.776, Y  +376.710, Z    +0.000, E1   +21.698, E3 +571579.813}
SPL {X  -162.707, Y  +374.438, Z    +0.000, E1   +21.688, E3 +571591.817}
SPL {X  -162.607, Y  +372.171, Z    +0.000, E1   +21.692, E3 +571603.617}
SPL {X  -162.494, Y  +370.197, Z    +0.000, E1   +21.655, E3 +571614.243}
SPL {X  -162.349, Y  +368.131, Z    +0.000, E1   +21.624, E3 +571625.361}
SPL {X  -162.161, Y  +365.866, Z    +0.000, E1   +21.642, E3 +571637.046}
SPL {X  -161.927, Y  +363.466, Z    +0.000, E1   +21.730, E3 +571648.818}
SPL {X  -160.290, Y  +351.907, Z    +0.000, E1   +27.562, E3 +571656.395}
SPL {X  -159.725, Y  +348.905, Z    +0.000, E1   +26.136, E3 +571681.631}
ENDSPLINE

SPLINE
SPL {X  -160.871, Y  +355.385, Z    +0.000, E1   +21.841, E3 +571690.474}
SPL {X  -161.833, Y  +362.603, Z    +0.000, E1   +17.021, E3 +571700.505}
ENDSPLINE

SPLINE
SPL {X  -160.786, Y  +354.842, Z    +0.000, E1   +19.274, E3 +571732.660}
ENDSPLINE

SPLINE
SPL {X  -162.485, Y  +370.062, Z    +0.000, E1   +10.606, E3 +571739.038}
SPL {X  -162.818, Y  +379.636, Z    +0.000, E1    +5.115, E3 +571728.387}
SPL {X  -162.820, Y  +386.976, Z    +0.000, E1    +0.144, E3 +571727.486}
SPL {X  -162.820, Y  +391.982, Z    +0.000, E1    -3.443, E3 +571734.251}
SPL {X  -162.820, Y  +399.630, Z    +0.000, E1    -9.426, E3 +571736.758}
SPL {X  -162.820, Y  +408.127, Z    +0.000, E1   -18.417, E3 +571723.047}
SPL {X  -162.820, Y  +420.083, Z    +0.000, E1   -24.325, E3 +571743.522}
SPL {X  -162.820, Y  +428.527, Z    +0.000, E1   -26.988, E3 +571760.814}
SPL {X  -162.820, Y  +431.191, Z    +0.000, E1   -23.548, E3 +571795.668}
SPL {X  -162.820, Y  +432.946, Z    +0.000, E1   -22.795, E3 +571810.071}
SPL {X  -162.820, Y  +434.888, Z    +0.000, E1   -22.823, E3 +571819.478}
SPL {X  -162.820, Y  +436.834, Z    +0.000, E1   -22.779, E3 +571829.438}
SPL {X  -162.820, Y  +438.868, Z    +0.000, E1   -22.837, E3 +571839.091}
SPL {X  -162.820, Y  +441.351, Z    +0.000, E1   -22.805, E3 +571851.667}
SPL {X  -162.820, Y  +443.809, Z    +0.000, E1   -22.804, E3 +571863.833}
SPL {X  -162.820, Y  +446.105, Z    +0.000, E1   -22.815, E3 +571875.075}
SPL {X  -162.820, Y  +447.974, Z    +0.000, E1   -22.856, E3 +571883.978}
SPL {X  -162.820, Y  +449.911, Z    +0.000, E1   -22.774, E3 +571894.253}
SPL {X  -162.820, Y  +451.861, Z    +0.000, E1   -22.750, E3 +571904.100}
SPL {X  -162.820, Y  +454.167, Z    +0.000, E1   -22.842, E3 +571914.830}
SPL {X  -162.820, Y  +456.529, Z    +0.000, E1   -22.855, E3 +571926.358}
SPL {X  -162.820, Y  +458.725, Z    +0.000, E1   -22.793, E3 +571937.763}
SPL {X  -162.820, Y  +461.700, Z    +0.000, E1   -22.822, E3 +571952.385}
SPL {X  -162.820, Y  +464.633, Z    +0.000, E1   -22.813, E3 +571966.882}
SPL {X  -162.820, Y  +466.699, Z    +0.000, E1   -22.824, E3 +571976.928}
SPL {X  -162.820, Y  +468.655, Z    +0.000, E1   -22.858, E3 +571986.372}
SPL {X  -162.820, Y  +470.892, Z    +0.000, E1   -22.837, E3 +571997.610}
SPL {X  -162.820, Y  +472.726, Z    +0.000, E1   -22.777, E3 +572007.149}
SPL {X  -162.820, Y  +475.118, Z    +0.000, E1   -22.777, E3 +572019.121}
SPL {X  -162.820, Y  +478.177, Z    +0.000, E1   -22.834, E3 +572033.813}
SPL {X  -162.820, Y  +481.034, Z    +0.000, E1   -22.831, E3 +572047.951}
SPL {X  -162.820, Y  +483.391, Z    +0.000, E1   -22.793, E3 +572059.887}
SPL {X  -162.820, Y  +486.307, Z    +0.000, E1   -22.833, E3 +572074.141}
SPL {X  -162.820, Y  +488.828, Z    +0.000, E1   -22.793, E3 +572086.784}
SPL {X  -162.820, Y  +491.768, Z    +0.000, E1   -22.852, E3 +572101.081}
SPL {X  -162.820, Y  +495.526, Z    +0.000, E1   -22.833, E3 +572119.852}
SPL {X  -162.820, Y  +499.330, Z    +0.000, E1   -22.841, E3 +572138.633}
SPL {X  -162.820, Y  +503.049, Z    +0.000, E1   -22.823, E3 +572157.182}
SPL {X  -162.820, Y  +506.908, Z    +0.000, E1   -22.877, E3 +572175.852}
SPL {X  -162.820, Y  +510.068, Z    +0.000, E1   -22.761, E3 +572192.324}
SPL {X  -162.820, Y  +512.359, Z    +0.000, E1   -22.823, E3 +572203.055}
SPL {X  -162.820, Y  +513.873, Z    +0.000, E1   -22.800, E3 +572210.742}
SPL {X  -162.820, Y  +516.100, Z    +0.000, E1   -22.809, E3 +572221.818}
SPL {X  -162.820, Y  +518.662, Z    +0.000, E1   -22.847, E3 +572234.117}
SPL {X  -162.820, Y  +520.641, Z    +0.000, E1   -22.790, E3 +572244.358}
SPL {X  -162.820, Y  +523.535, Z    +0.000, E1   -22.857, E3 +572258.327}
SPL {X  -162.820, Y  +526.661, Z    +0.000, E1   -22.801, E3 +572274.151}
SPL {X  -162.820, Y  +528.725, Z    +0.000, E1   -22.770, E3 +572284.520}
SPL {X  -162.820, Y  +530.303, Z    +0.000, E1   -22.798, E3 +572292.140}
SPL {X  -162.820, Y  +532.614, Z    +0.000, E1   -22.828, E3 +572303.408}
SPL {X  -162.820, Y  +534.838, Z    +0.000, E1   -22.864, E3 +572314.037}
SPL {X  -162.820, Y  +536.882, Z    +0.000, E1   -22.782, E3 +572324.892}
SPL {X  -162.820, Y  +539.194, Z    +0.000, E1   -22.826, E3 +572335.940}
SPL {X  -162.820, Y  +541.555, Z    +0.000, E1   -22.817, E3 +572347.755}
SPL {X  -162.820, Y  +543.728, Z    +0.000, E1   -22.799, E3 +572358.612}
SPL {X  -162.820, Y  +545.925, Z    +0.000, E1   -22.803, E3 +572369.482}
SPL {X  -162.820, Y  +549.071, Z    +0.000, E1   -22.836, E3 +572385.009}
SPL {X  -162.820, Y  +553.089, Z    +0.000, E1   -22.838, E3 +572404.909}
SPL {X  -162.820, Y  +556.430, Z    +0.000, E1   -22.821, E3 +572421.411}
SPL {X  -162.820, Y  +558.974, Z    +0.000, E1   -22.806, E3 +572434.111}
SPL {X  -162.820, Y  +562.171, Z    +0.000, E1   -22.845, E3 +572449.809}
SPL {X  -162.820, Y  +565.170, Z    +0.000, E1   -22.801, E3 +572464.822}
SPL {X  -162.820, Y  +567.308, Z    +0.000, E1   -22.750, E3 +572475.838}
SPL {X  -162.820, Y  +570.378, Z    +0.000, E1   -22.843, E3 +572490.462}
SPL {X  -162.820, Y  +573.634, Z    +0.000, E1   -22.827, E3 +572506.606}
SPL {X  -162.820, Y  +576.228, Z    +0.000, E1   -22.814, E3 +572519.502}
SPL {X  -162.820, Y  +578.553, Z    +0.000, E1   -22.801, E3 +572531.118}
SPL {X  -162.820, Y  +581.064, Z    +0.000, E1   -22.823, E3 +572543.402}
SPL {X  -162.820, Y  +583.435, Z    +0.000, E1   -22.808, E3 +572555.224}
SPL {X  -162.820, Y  +585.410, Z    +0.000, E1   -22.764, E3 +572565.360}
SPL {X  -162.820, Y  +587.676, Z    +0.000, E1   -22.853, E3 +572575.874}
SPL {X  -162.820, Y  +590.707, Z    +0.000, E1   -22.855, E3 +572591.025}
SPL {X  -162.820, Y  +593.650, Z    +0.000, E1   -22.810, E3 +572605.785}
SPL {X  -162.820, Y  +595.830, Z    +0.000, E1   -22.828, E3 +572616.401}
SPL {X  -162.820, Y  +598.094, Z    +0.000, E1   -22.843, E3 +572627.514}
SPL {X  -162.820, Y  +600.420, Z    +0.000, E1   -22.826, E3 +572639.145}
SPL {X  -162.820, Y  +602.573, Z    +0.000, E1   -22.830, E3 +572649.730}
SPL {X  -162.820, Y  +604.828, Z    +0.000, E1   -22.784, E3 +572661.369}
SPL {X  -162.820, Y  +608.133, Z    +0.000, E1   -22.831, E3 +572677.486}
SPL {X  -162.820, Y  +611.103, Z    +0.000, E1   -22.785, E3 +572692.412}
SPL {X  -162.820, Y  +613.294, Z    +0.000, E1   -22.780, E3 +572703.285}
SPL {X  -162.820, Y  +615.356, Z    +0.000, E1   -22.799, E3 +572713.342}
SPL {X  -162.820, Y  +617.439, Z    +0.000, E1   -22.808, E3 +572723.601}
SPL {X  -162.820, Y  +619.665, Z    +0.000, E1   -22.817, E3 +572734.569}
SPL {X  -162.820, Y  +621.733, Z    +0.000, E1   -22.759, E3 +572745.293}
SPL {X  -162.820, Y  +624.076, Z    +0.000, E1   -22.774, E3 +572756.798}
SPL {X  -162.820, Y  +627.244, Z    +0.000, E1   -22.803, E3 +572772.480}
SPL {X  -162.820, Y  +630.349, Z    +0.000, E1   -22.766, E3 +572788.012}
SPL {X  -162.820, Y  +632.572, Z    +0.000, E1   -22.785, E3 +572798.819}
SPL {X  -162.820, Y  +634.507, Z    +0.000, E1   -22.784, E3 +572808.458}
SPL {X  -162.820, Y  +636.863, Z    +0.000, E1   -22.760, E3 +572820.380}
SPL {X  -162.820, Y  +640.111, Z    +0.000, E1   -22.809, E3 +572836.262}
SPL {X  -162.820, Y  +643.449, Z    +0.000, E1   -22.796, E3 +572852.780}
SPL {X  -162.820, Y  +645.630, Z    +0.000, E1   -22.795, E3 +572863.476}
SPL {X  -162.820, Y  +647.561, Z    +0.000, E1   -22.705, E3 +572873.927}
SPL {X  -162.820, Y  +651.051, Z    +0.000, E1   -22.833, E3 +572890.346}
SPL {X  -162.820, Y  +653.898, Z    +0.000, E1   -22.796, E3 +572904.532}
SPL {X  -162.820, Y  +656.161, Z    +0.000, E1   -22.812, E3 +572915.654}
SPL {X  -162.820, Y  +658.384, Z    +0.000, E1   -22.822, E3 +572926.520}
SPL {X  -162.820, Y  +660.215, Z    +0.000, E1   -22.649, E3 +572937.111}
SPL {X  -162.820, Y  +662.823, Z    +0.000, E1   -22.799, E3 +572948.819}
SPL {X  -162.820, Y  +665.862, Z    +0.000, E1   -22.864, E3 +572963.518}
SPL {X  -162.820, Y  +668.960, Z    +0.000, E1   -22.773, E3 +572979.469}
SPL {X  -162.820, Y  +672.333, Z    +0.000, E1   -22.837, E3 +572995.805}
SPL {X  -162.812, Y  +675.071, Z    +0.000, E1   -22.742, E3 +573009.950}
SPL {X  -162.773, Y  +677.428, Z    +0.000, E1   -22.762, E3 +573021.548}
SPL {X  -162.691, Y  +679.987, Z    +0.000, E1   -22.794, E3 +573033.961}
SPL {X  -162.604, Y  +681.880, Z    +0.000, E1   -22.691, E3 +573044.122}
SPL {X  -162.458, Y  +684.346, Z    +0.000, E1   -22.764, E3 +573055.915}
SPL {X  -162.296, Y  +686.547, Z    +0.000, E1   -22.660, E3 +573067.532}
SPL {X  -162.090, Y  +688.902, Z    +0.000, E1   -22.700, E3 +573079.040}
SPL {X  -161.474, Y  +694.390, Z    +0.000, E1   -24.298, E3 +573092.395}
SPL {X  -158.730, Y  +709.763, Z    +0.000, E1   -31.225, E3 +573103.734}
ENDSPLINE

SPLINE
SPL {X  -160.932, Y  +698.225, Z    +0.000, E1   -21.712, E3 +573134.843}
SPL {X  -161.917, Y  +690.622, Z    +0.000, E1   -16.445, E3 +573148.444}
ENDSPLINE

SPLINE
SPL {X  -161.349, Y  +695.340, Z    +0.000, E1   -18.625, E3 +573156.063}
ENDSPLINE

SPLINE
SPL {X  -162.534, Y  +683.153, Z    +0.000, E1   -10.475, E3 +573177.193}
SPL {X  -162.820, Y  +667.630, Z    +0.000, E1    -0.882, E3 +573171.170}
SPL {X  -162.820, Y  +661.883, Z    +0.000, E1    +3.373, E3 +573176.613}
SPL {X  -162.820, Y  +653.808, Z    +0.000, E1    +9.891, E3 +573174.304}
SPL {X  -162.820, Y  +632.548, Z    +0.000, E1   +27.446, E3 +573170.841}
ENDSPLINE

SPLINE
SPL {X  -162.820, Y  +638.080, Z    +0.000, E1   +18.858, E3 +573198.589}
ENDSPLINE

SPLINE
SPL {X  -162.820, Y  +623.278, Z    +0.000, E1   +28.723, E3 +573200.160}
SPL {X  -162.820, Y  +618.658, Z    +0.000, E1   +26.841, E3 +573228.769}
ENDSPLINE

SPLINE
SPL {X  -162.820, Y  +623.685, Z    +0.000, E1   +22.346, E3 +573241.075}
ENDSPLINE

SPLINE
SPL {X  -162.820, Y  +621.304, Z    +0.000, E1   +22.259, E3 +573253.891}
SPL {X  -162.820, Y  +618.758, Z    +0.000, E1   +22.239, E3 +573267.041}
SPL {X  -162.820, Y  +616.062, Z    +0.000, E1   +22.275, E3 +573280.462}
SPL {X  -162.820, Y  +613.536, Z    +0.000, E1   +22.242, E3 +573293.584}
SPL {X  -162.820, Y  +610.461, Z    +0.000, E1   +22.264, E3 +573309.215}
SPL {X  -162.820, Y  +607.796, Z    +0.000, E1   +22.261, E3 +573322.586}
SPL {X  -162.820, Y  +605.178, Z    +0.000, E1   +22.267, E3 +573336.070}
SPL {X  -162.820, Y  +602.350, Z    +0.000, E1   +22.224, E3 +573350.687}
SPL {X  -162.820, Y  +599.842, Z    +0.000, E1   +22.298, E3 +573362.838}
SPL {X  -162.820, Y  +597.194, Z    +0.000, E1   +22.253, E3 +573376.759}
SPL {X  -162.820, Y  +594.779, Z    +0.000, E1   +22.284, E3 +573388.663}
SPL {X  -162.820, Y  +592.389, Z    +0.000, E1   +22.245, E3 +573401.280}
SPL {X  -162.820, Y  +589.492, Z    +0.000, E1   +22.304, E3 +573415.464}
SPL {X  -162.820, Y  +587.447, Z    +0.000, E1   +22.279, E3 +573425.993}
SPL {X  -162.820, Y  +585.192, Z    +0.000, E1   +22.298, E3 +573437.403}
SPL {X  -162.820, Y  +582.610, Z    +0.000, E1   +22.234, E3 +573451.027}
SPL {X  -162.820, Y  +580.317, Z    +0.000, E1   +22.300, E3 +573462.081}
SPL {X  -162.820, Y  +578.878, Z    +0.000, E1   +22.272, E3 +573469.590}
SPL {X  -162.820, Y  +576.856, Z    +0.000, E1   +22.233, E3 +573480.349}
SPL {X  -162.820, Y  +574.811, Z    +0.000, E1   +22.236, E3 +573490.612}
SPL {X  -162.820, Y  +572.645, Z    +0.000, E1   +22.246, E3 +573501.708}
SPL {X  -162.820, Y  +570.282, Z    +0.000, E1   +22.231, E3 +573513.758}
SPL {X  -162.820, Y  +567.961, Z    +0.000, E1   +22.247, E3 +573525.548}
SPL {X  -162.820, Y  +564.506, Z    +0.000, E1   +22.298, E3 +573542.862}
SPL {X  -162.820, Y  +561.620, Z    +0.000, E1   +22.191, E3 +573558.243}
SPL {X  -162.820, Y  +559.515, Z    +0.000, E1   +22.273, E3 +573568.245}
SPL {X  -162.820, Y  +556.723, Z    +0.000, E1   +22.309, E3 +573582.328}
SPL {X  -162.820, Y  +554.378, Z    +0.000, E1   +22.288, E3 +573594.174}
SPL {X  -162.820, Y  +552.787, Z    +0.000, E1   +22.213, E3 +573602.996}
SPL {X  -162.820, Y  +550.871, Z    +0.000, E1   +22.229, E3 +573612.590}
SPL {X  -162.820, Y  +548.168, Z    +0.000, E1   +22.298, E3 +573625.926}
SPL {X  -162.820, Y  +545.860, Z    +0.000, E1   +22.216, E3 +573638.184}
SPL {X  -162.820, Y  +543.558, Z    +0.000, E1   +22.285, E3 +573649.414}
SPL {X  -162.820, Y  +541.633, Z    +0.000, E1   +22.257, E3 +573659.342}
SPL {X  -162.820, Y  +539.116, Z    +0.000, E1   +22.302, E3 +573671.953}
SPL {X  -162.820, Y  +535.523, Z    +0.000, E1   +22.266, E3 +573690.615}
SPL {X  -162.820, Y  +531.757, Z    +0.000, E1   +22.276, E3 +573709.669}
SPL {X  -162.820, Y  +527.980, Z    +0.000, E1   +22.326, E3 +573728.500}
SPL {X  -162.820, Y  +524.599, Z    +0.000, E1   +22.287, E3 +573745.898}
SPL {X  -162.820, Y  +522.011, Z    +0.000, E1   +22.282, E3 +573758.975}
SPL {X  -162.820, Y  +519.457, Z    +0.000, E1   +22.481, E3 +573770.264}
SPL {X  -162.820, Y  +506.285, Z    +0.000, E1   +28.538, E3 +573781.722}
SPL {X  -162.820, Y  +504.441, Z    +0.000, E1   +27.574, E3 +573796.064}
SPL {X  -162.820, Y  +502.813, Z    +0.000, E1   +26.013, E3 +573814.262}
SPL {X  -162.820, Y  +502.016, Z    +0.000, E1   +24.802, E3 +573826.604}
SPL {X  -162.820, Y  +501.060, Z    +0.000, E1   +24.081, E3 +573836.794}
SPL {X  -162.820, Y  +500.336, Z    +0.000, E1   +23.110, E3 +573847.934}
SPL {X  -162.820, Y  +499.240, Z    +0.000, E1   +22.316, E3 +573860.244}
SPL {X  -162.820, Y  +498.027, Z    +0.000, E1   +21.516, E3 +573873.152}
SPL {X  -162.820, Y  +495.897, Z    +0.000, E1   +21.662, E3 +573883.072}
SPL {X  -162.820, Y  +493.717, Z    +0.000, E1   +21.704, E3 +573894.179}
SPL {X  -162.820, Y  +491.396, Z    +0.000, E1   +21.707, E3 +573906.303}
SPL {X  -162.820, Y  +488.560, Z    +0.000, E1   +21.695, E3 +573921.412}
SPL {X  -162.820, Y  +485.661, Z    +0.000, E1   +21.712, E3 +573936.297}
SPL {X  -162.820, Y  +483.668, Z    +0.000, E1   +21.664, E3 +573947.125}
SPL {X  -162.820, Y  +481.739, Z    +0.000, E1   +21.704, E3 +573956.839}
SPL {X  -162.820, Y  +479.894, Z    +0.000, E1   +21.695, E3 +573966.626}
SPL {X  -162.820, Y  +477.685, Z    +0.000, E1   +21.656, E3 +573978.563}
SPL {X  -162.820, Y  +475.419, Z    +0.000, E1   +21.711, E3 +573989.916}
SPL {X  -162.820, Y  +473.301, Z    +0.000, E1   +21.712, E3 +574001.013}
SPL {X  -162.820, Y  +470.965, Z    +0.000, E1   +21.700, E3 +574013.358}
SPL {X  -162.820, Y  +469.036, Z    +0.000, E1   +21.695, E3 +574023.402}
SPL {X  -162.820, Y  +467.138, Z    +0.000, E1   +21.678, E3 +574033.573}
SPL {X  -162.820, Y  +465.011, Z    +0.000, E1   +21.692, E3 +574044.556}
SPL {X  -162.820, Y  +462.669, Z    +0.000, E1   +21.752, E3 +574056.337}
SPL {X  -162.820, Y  +460.725, Z    +0.000, E1   +21.689, E3 +574066.950}
SPL {X  -162.820, Y  +458.666, Z    +0.000, E1   +21.695, E3 +574077.762}
SPL {X  -162.820, Y  +456.431, Z    +0.000, E1   +21.708, E3 +574089.290}
SPL {X  -162.820, Y  +453.609, Z    +0.000, E1   +21.757, E3 +574103.824}
SPL {X  -162.820, Y  +450.610, Z    +0.000, E1   +21.698, E3 +574119.881}
SPL {X  -162.820, Y  +448.170, Z    +0.000, E1   +21.667, E3 +574132.902}
SPL {X  -162.820, Y  +446.246, Z    +0.000, E1   +21.696, E3 +574142.720}
SPL {X  -162.820, Y  +443.784, Z    +0.000, E1   +21.713, E3 +574155.506}
SPL {X  -162.820, Y  +440.567, Z    +0.000, E1   +21.731, E3 +574172.346}
SPL {X  -162.820, Y  +437.628, Z    +0.000, E1   +21.678, E3 +574188.010}
SPL {X  -162.820, Y  +434.473, Z    +0.000, E1   +21.747, E3 +574204.106}
SPL {X  -162.820, Y  +431.492, Z    +0.000, E1   +21.686, E3 +574220.055}
SPL {X  -162.820, Y  +429.074, Z    +0.000, E1   +21.710, E3 +574232.507}
SPL {X  -162.820, Y  +426.023, Z    +0.000, E1   +21.718, E3 +574248.575}
SPL {X  -162.820, Y  +422.986, Z    +0.000, E1   +21.685, E3 +574264.622}
SPL {X  -162.820, Y  +420.528, Z    +0.000, E1   +21.706, E3 +574277.272}
SPL {X  -162.820, Y  +418.116, Z    +0.000, E1   +21.761, E3 +574289.419}
SPL {X  -162.820, Y  +416.127, Z    +0.000, E1   +21.715, E3 +574300.125}
SPL {X  -162.820, Y  +414.361, Z    +0.000, E1   +21.613, E3 +574310.312}
SPL {X  -162.820, Y  +412.134, Z    +0.000, E1   +21.697, E3 +574321.256}
SPL {X  -162.820, Y  +409.248, Z    +0.000, E1   +21.741, E3 +574336.192}
SPL {X  -162.820, Y  +406.238, Z    +0.000, E1   +21.697, E3 +574352.160}
SPL {X  -162.820, Y  +404.001, Z    +0.000, E1   +21.723, E3 +574363.589}
SPL {X  -162.820, Y  +402.223, Z    +0.000, E1   +21.697, E3 +574373.075}
SPL {X  -162.820, Y  +400.348, Z    +0.000, E1   +21.713, E3 +574382.800}
SPL {X  -162.820, Y  +398.298, Z    +0.000, E1   +21.721, E3 +574393.416}
SPL {X  -162.820, Y  +396.371, Z    +0.000, E1   +21.713, E3 +574403.598}
SPL {X  -162.820, Y  +394.508, Z    +0.000, E1   +21.616, E3 +574414.153}
SPL {X  -162.820, Y  +392.435, Z    +0.000, E1   +21.681, E3 +574424.507}
SPL {X  -162.820, Y  +389.390, Z    +0.000, E1   +21.742, E3 +574440.113}
SPL {X  -162.820, Y  +386.818, Z    +0.000, E1   +21.679, E3 +574453.872}
SPL {X  -162.820, Y  +384.697, Z    +0.000, E1   +21.693, E3 +574464.942}
SPL {X  -162.820, Y  +382.288, Z    +0.000, E1   +21.742, E3 +574477.066}
SPL {X  -162.820, Y  +380.381, Z    +0.000, E1   +21.655, E3 +574487.791}
SPL {X  -162.808, Y  +378.512, Z    +0.000, E1   +21.736, E3 +574496.843}
SPL {X  -162.776, Y  +376.710, Z    +0.000, E1   +21.698, E3 +574506.643}
SPL {X  -162.707, Y  +374.438, Z    +0.000, E1   +21.688, E3 +574518.646}
SPL {X  -162.607, Y  +372.171, Z    +0.000, E1   +21.692, E3 +574530.446}
SPL {X  -162.494, Y  +370.197, Z    +0.000, E1   +21.655, E3 +574541.072}
SPL {X  -162.349, Y  +368.131, Z    +0.000, E1   +21.624, E3 +574552.190}
SPL {X  -162.161, Y  +365.866, Z    +0.000, E1   +21.642, E3 +574563.876}
SPL {X  -161.927, Y  +363.466, Z    +0.000, E1   +21.730, E3 +574575.647}
SPL {X  -160.290, Y  +351.907, Z    +0.000, E1   +27.562, E3 +574583.225}
SPL {X  -159.725, Y  +348.905, Z    +0.000, E1   +26.136, E3 +574608.460}
ENDSPLINE

SPLINE
SPL {X  -160.871, Y  +355.385, Z    +0.000, E1   +21.841, E3 +574617.303}
SPL {X  -161.833, Y  +362.603, Z    +0.000, E1   +17.021, E3 +574627.334}
ENDSPLINE

SPLINE
SPL {X  -160.786, Y  +354.842, Z    +0.000, E1   +19.274, E3 +574659.489}
ENDSPLINE

SPLINE
SPL {X  -162.485, Y  +370.062, Z    +0.000, E1   +10.606, E3 +574665.868}
SPL {X  -162.818, Y  +379.636, Z    +0.000, E1    +5.115, E3 +574655.216}
SPL {X  -162.820, Y  +386.976, Z    +0.000, E1    +0.144, E3 +574654.316}
SPL {X  -162.820, Y  +390.236, Z    +0.000, E1    -2.204, E3 +574660.374}
SPL {X  -162.820, Y  +393.415, Z    +0.000, E1    -4.587, E3 +574661.658}
SPL {X  -162.820, Y  +399.630, Z    +0.000, E1    -9.426, E3 +574663.588}
SPL {X  -162.820, Y  +408.127, Z    +0.000, E1   -18.417, E3 +574649.876}
SPL {X  -162.820, Y  +420.083, Z    +0.000, E1   -24.325, E3 +574670.352}
SPL {X  -162.820, Y  +428.527, Z    +0.000, E1   -26.988, E3 +574687.644}
SPL {X  -162.820, Y  +431.191, Z    +0.000, E1   -23.548, E3 +574722.497}
SPL {X  -162.820, Y  +432.946, Z    +0.000, E1   -22.795, E3 +574736.900}
SPL {X  -162.820, Y  +434.888, Z    +0.000, E1   -22.823, E3 +574746.307}
SPL {X  -162.820, Y  +436.834, Z    +0.000, E1   -22.779, E3 +574756.267}
SPL {X  -162.820, Y  +438.868, Z    +0.000, E1   -22.837, E3 +574765.921}
SPL {X  -162.820, Y  +441.351, Z    +0.000, E1   -22.805, E3 +574778.496}
SPL {X  -162.820, Y  +443.809, Z    +0.000, E1   -22.804, E3 +574790.662}
SPL {X  -162.820, Y  +446.105, Z    +0.000, E1   -22.815, E3 +574801.905}
SPL {X  -162.820, Y  +447.974, Z    +0.000, E1   -22.856, E3 +574810.807}
SPL {X  -162.820, Y  +449.911, Z    +0.000, E1   -22.774, E3 +574821.082}
SPL {X  -162.820, Y  +451.861, Z    +0.000, E1   -22.750, E3 +574830.930}
SPL {X  -162.820, Y  +454.167, Z    +0.000, E1   -22.842, E3 +574841.659}
SPL {X  -162.820, Y  +456.529, Z    +0.000, E1   -22.855, E3 +574853.188}
SPL {X  -162.820, Y  +458.725, Z    +0.000, E1   -22.793, E3 +574864.592}
SPL {X  -162.820, Y  +461.700, Z    +0.000, E1   -22.822, E3 +574879.214}
SPL {X  -162.820, Y  +464.633, Z    +0.000, E1   -22.813, E3 +574893.711}
SPL {X  -162.820, Y  +466.699, Z    +0.000, E1   -22.824, E3 +574903.757}
SPL {X  -162.820, Y  +468.655, Z    +0.000, E1   -22.858, E3 +574913.201}
SPL {X  -162.820, Y  +470.892, Z    +0.000, E1   -22.837, E3 +574924.440}
SPL {X  -162.820, Y  +473.485, Z    +0.000, E1   -22.806, E3 +574937.638}
SPL {X  -162.820, Y  +476.589, Z    +0.000, E1   -22.788, E3 +574953.160}
SPL {X  -162.820, Y  +478.914, Z    +0.000, E1   -22.821, E3 +574964.258}
SPL {X  -162.820, Y  +481.034, Z    +0.000, E1   -22.831, E3 +574974.780}
SPL {X  -162.820, Y  +484.256, Z    +0.000, E1   -22.840, E3 +574990.799}
SPL {X  -162.820, Y  +487.952, Z    +0.000, E1   -22.824, E3 +575009.229}
SPL {X  -162.820, Y  +491.768, Z    +0.000, E1   -22.852, E3 +575027.910}
SPL {X  -162.820, Y  +495.526, Z    +0.000, E1   -22.833, E3 +575046.681}
SPL {X  -162.820, Y  +499.330, Z    +0.000, E1   -22.841, E3 +575065.462}
SPL {X  -162.820, Y  +503.049, Z    +0.000, E1   -22.823, E3 +575084.012}
SPL {X  -162.820, Y  +506.908, Z    +0.000, E1   -22.877, E3 +575102.682}
SPL {X  -162.820, Y  +510.068, Z    +0.000, E1   -22.761, E3 +575119.153}
SPL {X  -162.820, Y  +512.359, Z    +0.000, E1   -22.823, E3 +575129.885}
SPL {X  -162.820, Y  +513.873, Z    +0.000, E1   -22.800, E3 +575137.571}
SPL {X  -162.820, Y  +516.100, Z    +0.000, E1   -22.809, E3 +575148.648}
SPL {X  -162.820, Y  +518.662, Z    +0.000, E1   -22.847, E3 +575160.946}
SPL {X  -162.820, Y  +520.641, Z    +0.000, E1   -22.790, E3 +575171.187}
SPL {X  -162.820, Y  +523.535, Z    +0.000, E1   -22.857, E3 +575185.156}
SPL {X  -162.820, Y  +526.661, Z    +0.000, E1   -22.801, E3 +575200.980}
SPL {X  -162.820, Y  +528.725, Z    +0.000, E1   -22.770, E3 +575211.350}
SPL {X  -162.820, Y  +530.303, Z    +0.000, E1   -22.798, E3 +575218.969}
SPL {X  -162.820, Y  +532.614, Z    +0.000, E1   -22.828, E3 +575230.237}
SPL {X  -162.820, Y  +534.838, Z    +0.000, E1   -22.864, E3 +575240.866}
SPL {X  -162.820, Y  +536.882, Z    +0.000, E1   -22.782, E3 +575251.721}
SPL {X  -162.820, Y  +539.194, Z    +0.000, E1   -22.826, E3 +575262.769}
SPL {X  -162.820, Y  +541.555, Z    +0.000, E1   -22.817, E3 +575274.584}
SPL {X  -162.820, Y  +543.728, Z    +0.000, E1   -22.799, E3 +575285.441}
SPL {X  -162.820, Y  +545.925, Z    +0.000, E1   -22.803, E3 +575296.311}
SPL {X  -162.820, Y  +548.328, Z    +0.000, E1   -22.796, E3 +575308.307}
SPL {X  -162.820, Y  +551.027, Z    +0.000, E1   -22.819, E3 +575321.500}
SPL {X  -162.820, Y  +553.721, Z    +0.000, E1   -22.807, E3 +575334.944}
SPL {X  -162.820, Y  +556.430, Z    +0.000, E1   -22.821, E3 +575348.240}
SPL {X  -162.820, Y  +559.675, Z    +0.000, E1   -22.837, E3 +575364.320}
SPL {X  -162.820, Y  +562.799, Z    +0.000, E1   -22.814, E3 +575379.826}
SPL {X  -162.820, Y  +565.170, Z    +0.000, E1   -22.801, E3 +575391.651}
SPL {X  -162.820, Y  +568.020, Z    +0.000, E1   -22.787, E3 +575406.038}
SPL {X  -162.820, Y  +570.992, Z    +0.000, E1   -22.834, E3 +575420.257}
SPL {X  -162.820, Y  +572.901, Z    +0.000, E1   -22.775, E3 +575430.125}
SPL {X  -162.820, Y  +575.638, Z    +0.000, E1   -22.855, E3 +575443.235}
SPL {X  -162.820, Y  +578.553, Z    +0.000, E1   -22.801, E3 +575457.947}
SPL {X  -162.820, Y  +581.064, Z    +0.000, E1   -22.823, E3 +575470.232}
SPL {X  -162.820, Y  +583.435, Z    +0.000, E1   -22.808, E3 +575482.053}
SPL {X  -162.820, Y  +585.410, Z    +0.000, E1   -22.764, E3 +575492.189}
SPL {X  -162.820, Y  +587.676, Z    +0.000, E1   -22.853, E3 +575502.704}
SPL {X  -162.820, Y  +589.682, Z    +0.000, E1   -22.776, E3 +575513.234}
SPL {X  -162.820, Y  +591.720, Z    +0.000, E1   -22.868, E3 +575522.544}
SPL {X  -162.820, Y  +593.650, Z    +0.000, E1   -22.810, E3 +575532.614}
SPL {X  -162.820, Y  +595.830, Z    +0.000, E1   -22.828, E3 +575543.230}
SPL {X  -162.820, Y  +598.094, Z    +0.000, E1   -22.843, E3 +575554.343}
SPL {X  -162.820, Y  +600.420, Z    +0.000, E1   -22.826, E3 +575565.974}
SPL {X  -162.820, Y  +602.573, Z    +0.000, E1   -22.830, E3 +575576.560}
SPL {X  -162.820, Y  +604.828, Z    +0.000, E1   -22.784, E3 +575588.198}
SPL {X  -162.820, Y  +607.142, Z    +0.000, E1   -22.808, E3 +575599.379}
SPL {X  -162.820, Y  +608.890, Z    +0.000, E1   -22.790, E3 +575608.203}
SPL {X  -162.820, Y  +611.103, Z    +0.000, E1   -22.785, E3 +575619.241}
SPL {X  -162.820, Y  +613.294, Z    +0.000, E1   -22.780, E3 +575630.115}
SPL {X  -162.820, Y  +615.356, Z    +0.000, E1   -22.799, E3 +575640.172}
SPL {X  -162.820, Y  +617.439, Z    +0.000, E1   -22.808, E3 +575650.430}
SPL {X  -162.820, Y  +619.665, Z    +0.000, E1   -22.817, E3 +575661.398}
SPL {X  -162.820, Y  +621.733, Z    +0.000, E1   -22.759, E3 +575672.122}
SPL {X  -162.820, Y  +624.076, Z    +0.000, E1   -22.774, E3 +575683.627}
SPL {X  -162.820, Y  +626.527, Z    +0.000, E1   -22.768, E3 +575695.870}
SPL {X  -162.820, Y  +629.758, Z    +0.000, E1   -22.800, E3 +575711.799}
SPL {X  -162.820, Y  +632.572, Z    +0.000, E1   -22.785, E3 +575725.648}
SPL {X  -162.820, Y  +634.507, Z    +0.000, E1   -22.784, E3 +575735.287}
SPL {X  -162.820, Y  +636.863, Z    +0.000, E1   -22.760, E3 +575747.209}
SPL {X  -162.820, Y  +639.254, Z    +0.000, E1   -22.767, E3 +575758.992}
SPL {X  -162.820, Y  +641.888, Z    +0.000, E1   -22.790, E3 +575771.939}
SPL {X  -162.820, Y  +644.915, Z    +0.000, E1   -22.818, E3 +575786.714}
SPL {X  -162.820, Y  +647.561, Z    +0.000, E1   -22.705, E3 +575800.756}
SPL {X  -162.820, Y  +649.758, Z    +0.000, E1   -22.780, E3 +575810.946}
SPL {X  -162.820, Y  +651.708, Z    +0.000, E1   -22.810, E3 +575820.441}
SPL {X  -162.820, Y  +653.898, Z    +0.000, E1   -22.796, E3 +575831.362}
SPL {X  -162.820, Y  +656.161, Z    +0.000, E1   -22.812, E3 +575842.483}
SPL {X  -162.820, Y  +658.384, Z    +0.000, E1   -22.822, E3 +575853.349}
SPL {X  -162.820, Y  +660.215, Z    +0.000, E1   -22.649, E3 +575863.940}
SPL {X  -162.820, Y  +662.823, Z    +0.000, E1   -22.799, E3 +575875.648}
SPL {X  -162.820, Y  +665.862, Z    +0.000, E1   -22.864, E3 +575890.347}
SPL {X  -162.820, Y  +668.960, Z    +0.000, E1   -22.773, E3 +575906.298}
SPL {X  -162.820, Y  +672.333, Z    +0.000, E1   -22.837, E3 +575922.634}
SPL {X  -162.812, Y  +675.071, Z    +0.000, E1   -22.742, E3 +575936.779}
SPL {X  -162.773, Y  +677.428, Z    +0.000, E1   -22.762, E3 +575948.377}
SPL {X  -162.691, Y  +679.987, Z    +0.000, E1   -22.794, E3 +575960.790}
SPL {X  -162.604, Y  +681.880, Z    +0.000, E1   -22.691, E3 +575970.951}
SPL {X  -162.458, Y  +684.346, Z    +0.000, E1   -22.764, E3 +575982.745}
SPL {X  -162.296, Y  +686.547, Z    +0.000, E1   -22.660, E3 +575994.361}
SPL {X  -162.090, Y  +688.902, Z    +0.000, E1   -22.700, E3 +576005.870}
SPL {X  -161.474, Y  +694.390, Z    +0.000, E1   -24.298, E3 +576019.225}
SPL {X  -158.553, Y  +710.529, Z    +0.000, E1   -30.890, E3 +576035.787}
ENDSPLINE

SPLINE
SPL {X  -161.215, Y  +696.305, Z    +0.000, E1   -20.575, E3 +576062.367}
SPL {X  -161.691, Y  +692.643, Z    +0.000, E1   -17.369, E3 +576078.555}
SPL {X  -162.534, Y  +683.153, Z    +0.000, E1   -10.475, E3 +576104.023}
SPL {X  -162.820, Y  +667.630, Z    +0.000, E1    -0.882, E3 +576097.999}
SPL {X  -162.820, Y  +661.883, Z    +0.000, E1    +3.373, E3 +576103.442}
SPL {X  -162.820, Y  +653.808, Z    +0.000, E1    +9.891, E3 +576101.133}
SPL {X  -162.820, Y  +632.548, Z    +0.000, E1   +27.446, E3 +576097.670}
ENDSPLINE

SPLINE
SPL {X  -162.820, Y  +638.080, Z    +0.000, E1   +18.858, E3 +576125.419}
ENDSPLINE

SPLINE
SPL {X  -162.820, Y  +623.278, Z    +0.000, E1   +28.723, E3 +576126.989}
SPL {X  -162.820, Y  +618.658, Z    +0.000, E1   +26.841, E3 +576155.598}
ENDSPLINE

SPLINE
SPL {X  -162.820, Y  +623.685, Z    +0.000, E1   +22.346, E3 +576167.905}
ENDSPLINE

SPLINE
SPL {X  -162.820, Y  +621.304, Z    +0.000, E1   +22.259, E3 +576180.720}
SPL {X  -162.820, Y  +618.758, Z    +0.000, E1   +22.239, E3 +576193.871}
SPL {X  -162.820, Y  +616.062, Z    +0.000, E1   +22.275, E3 +576207.291}
SPL {X  -162.820, Y  +613.536, Z    +0.000, E1   +22.242, E3 +576220.413}
SPL {X  -162.820, Y  +611.128, Z    +0.000, E1   +22.252, E3 +576232.584}
SPL {X  -162.820, Y  +608.428, Z    +0.000, E1   +22.255, E3 +576246.367}
SPL {X  -162.820, Y  +605.984, Z    +0.000, E1   +22.221, E3 +576259.004}
SPL {X  -162.820, Y  +603.020, Z    +0.000, E1   +22.272, E3 +576273.902}
SPL {X  -162.820, Y  +599.168, Z    +0.000, E1   +22.310, E3 +576293.170}
SPL {X  -162.820, Y  +596.569, Z    +0.000, E1   +22.222, E3 +576306.892}
SPL {X  -162.820, Y  +594.115, Z    +0.000, E1   +22.273, E3 +576319.118}
SPL {X  -162.820, Y  +591.721, Z    +0.000, E1   +22.239, E3 +576331.433}
SPL {X  -162.820, Y  +589.492, Z    +0.000, E1   +22.304, E3 +576342.294}
SPL {X  -162.820, Y  +587.447, Z    +0.000, E1   +22.279, E3 +576352.822}
SPL {X  -162.820, Y  +585.192, Z    +0.000, E1   +22.298, E3 +576364.233}
SPL {X  -162.820, Y  +582.610, Z    +0.000, E1   +22.234, E3 +576377.856}
SPL {X  -162.820, Y  +580.317, Z    +0.000, E1   +22.300, E3 +576388.910}
SPL {X  -162.820, Y  +578.878, Z    +0.000, E1   +22.272, E3 +576396.419}
SPL {X  -162.820, Y  +576.856, Z    +0.000, E1   +22.233, E3 +576407.178}
SPL {X  -162.820, Y  +573.830, Z    +0.000, E1   +22.272, E3 +576422.314}
SPL {X  -162.820, Y  +570.852, Z    +0.000, E1   +22.234, E3 +576437.773}
SPL {X  -162.820, Y  +568.608, Z    +0.000, E1   +22.253, E3 +576448.907}
SPL {X  -162.820, Y  +565.838, Z    +0.000, E1   +22.271, E3 +576463.138}
SPL {X  -162.820, Y  +562.162, Z    +0.000, E1   +22.252, E3 +576481.955}
SPL {X  -162.820, Y  +558.919, Z    +0.000, E1   +22.286, E3 +576498.118}
SPL {X  -162.820, Y  +555.548, Z    +0.000, E1   +22.322, E3 +576515.027}
SPL {X  -162.820, Y  +552.787, Z    +0.000, E1   +22.213, E3 +576529.825}
SPL {X  -162.820, Y  +550.136, Z    +0.000, E1   +22.258, E3 +576543.058}
SPL {X  -162.820, Y  +546.694, Z    +0.000, E1   +22.290, E3 +576560.381}
SPL {X  -162.820, Y  +543.558, Z    +0.000, E1   +22.285, E3 +576576.243}
SPL {X  -162.820, Y  +541.633, Z    +0.000, E1   +22.257, E3 +576586.172}
SPL {X  -162.820, Y  +539.116, Z    +0.000, E1   +22.302, E3 +576598.782}
SPL {X  -162.820, Y  +536.913, Z    +0.000, E1   +22.192, E3 +576610.707}
SPL {X  -162.820, Y  +534.880, Z    +0.000, E1   +22.252, E3 +576620.660}
SPL {X  -162.820, Y  +532.896, Z    +0.000, E1   +22.234, E3 +576630.821}
SPL {X  -162.820, Y  +531.056, Z    +0.000, E1   +22.251, E3 +576640.102}
SPL {X  -162.820, Y  +528.708, Z    +0.000, E1   +22.319, E3 +576651.484}
SPL {X  -162.820, Y  +525.932, Z    +0.000, E1   +22.258, E3 +576666.240}
SPL {X  -162.820, Y  +522.524, Z    +0.000, E1   +22.326, E3 +576682.964}
SPL {X  -162.820, Y  +519.457, Z    +0.000, E1   +22.481, E3 +576697.093}
SPL {X  -162.820, Y  +506.285, Z    +0.000, E1   +28.538, E3 +576708.551}
SPL {X  -162.820, Y  +504.441, Z    +0.000, E1   +27.574, E3 +576722.893}
SPL {X  -162.820, Y  +502.813, Z    +0.000, E1   +26.013, E3 +576741.091}
SPL {X  -162.820, Y  +502.016, Z    +0.000, E1   +24.802, E3 +576753.434}
SPL {X  -162.820, Y  +501.060, Z    +0.000, E1   +24.081, E3 +576763.623}
SPL {X  -162.820, Y  +499.934, Z    +0.000, E1   +22.814, E3 +576779.492}
SPL {X  -162.820, Y  +498.303, Z    +0.000, E1   +21.749, E3 +576796.748}
SPL {X  -162.820, Y  +495.897, Z    +0.000, E1   +21.662, E3 +576809.902}
SPL {X  -162.820, Y  +493.717, Z    +0.000, E1   +21.704, E3 +576821.008}
SPL {X  -162.820, Y  +491.396, Z    +0.000, E1   +21.707, E3 +576833.132}
SPL {X  -162.820, Y  +489.485, Z    +0.000, E1   +21.661, E3 +576843.480}
SPL {X  -162.820, Y  +487.723, Z    +0.000, E1   +21.665, E3 +576852.683}
SPL {X  -162.820, Y  +485.661, Z    +0.000, E1   +21.712, E3 +576863.127}
SPL {X  -162.820, Y  +482.775, Z    +0.000, E1   +21.716, E3 +576878.379}
SPL {X  -162.820, Y  +479.894, Z    +0.000, E1   +21.695, E3 +576893.455}
SPL {X  -162.820, Y  +477.685, Z    +0.000, E1   +21.656, E3 +576905.393}
SPL {X  -162.820, Y  +475.419, Z    +0.000, E1   +21.711, E3 +576916.745}
SPL {X  -162.820, Y  +473.301, Z    +0.000, E1   +21.712, E3 +576927.842}
SPL {X  -162.820, Y  +470.965, Z    +0.000, E1   +21.700, E3 +576940.187}
SPL {X  -162.820, Y  +469.036, Z    +0.000, E1   +21.695, E3 +576950.231}
SPL {X  -162.820, Y  +467.138, Z    +0.000, E1   +21.678, E3 +576960.403}
SPL {X  -162.820, Y  +465.011, Z    +0.000, E1   +21.692, E3 +576971.385}
SPL {X  -162.820, Y  +462.669, Z    +0.000, E1   +21.752, E3 +576983.166}
SPL {X  -162.820, Y  +460.725, Z    +0.000, E1   +21.689, E3 +576993.779}
SPL {X  -162.820, Y  +458.666, Z    +0.000, E1   +21.695, E3 +577004.591}
SPL {X  -162.820, Y  +456.431, Z    +0.000, E1   +21.708, E3 +577016.119}
SPL {X  -162.820, Y  +454.628, Z    +0.000, E1   +21.674, E3 +577025.838}
SPL {X  -162.820, Y  +452.690, Z    +0.000, E1   +21.773, E3 +577035.112}
SPL {X  -162.820, Y  +450.610, Z    +0.000, E1   +21.698, E3 +577046.710}
SPL {X  -162.820, Y  +448.170, Z    +0.000, E1   +21.667, E3 +577059.731}
SPL {X  -162.820, Y  +445.508, Z    +0.000, E1   +21.732, E3 +577073.250}
SPL {X  -162.820, Y  +442.443, Z    +0.000, E1   +21.712, E3 +577089.370}
SPL {X  -162.820, Y  +439.933, Z    +0.000, E1   +21.690, E3 +577102.651}
SPL {X  -162.820, Y  +437.628, Z    +0.000, E1   +21.678, E3 +577114.839}
SPL {X  -162.820, Y  +434.473, Z    +0.000, E1   +21.747, E3 +577130.935}
SPL {X  -162.820, Y  +431.492, Z    +0.000, E1   +21.686, E3 +577146.884}
SPL {X  -162.820, Y  +429.074, Z    +0.000, E1   +21.710, E3 +577159.336}
SPL {X  -162.820, Y  +426.023, Z    +0.000, E1   +21.718, E3 +577175.404}
SPL {X  -162.820, Y  +422.986, Z    +0.000, E1   +21.685, E3 +577191.451}
SPL {X  -162.820, Y  +420.528, Z    +0.000, E1   +21.706, E3 +577204.101}
SPL {X  -162.820, Y  +418.116, Z    +0.000, E1   +21.761, E3 +577216.249}
SPL {X  -162.820, Y  +416.127, Z    +0.000, E1   +21.715, E3 +577226.954}
SPL {X  -162.820, Y  +414.361, Z    +0.000, E1   +21.613, E3 +577237.141}
SPL {X  -162.820, Y  +411.450, Z    +0.000, E1   +21.710, E3 +577251.715}
SPL {X  -162.820, Y  +408.590, Z    +0.000, E1   +21.735, E3 +577266.340}
SPL {X  -162.820, Y  +406.238, Z    +0.000, E1   +21.697, E3 +577278.989}
SPL {X  -162.820, Y  +403.166, Z    +0.000, E1   +21.746, E3 +577294.795}
SPL {X  -162.820, Y  +400.348, Z    +0.000, E1   +21.713, E3 +577309.630}
SPL {X  -162.820, Y  +398.298, Z    +0.000, E1   +21.721, E3 +577320.245}
SPL {X  -162.820, Y  +396.371, Z    +0.000, E1   +21.713, E3 +577330.427}
SPL {X  -162.820, Y  +394.508, Z    +0.000, E1   +21.616, E3 +577340.982}
SPL {X  -162.820, Y  +391.777, Z    +0.000, E1   +21.714, E3 +577354.642}
SPL {X  -162.820, Y  +388.822, Z    +0.000, E1   +21.717, E3 +577369.962}
SPL {X  -162.820, Y  +386.818, Z    +0.000, E1   +21.679, E3 +577380.701}
SPL {X  -162.820, Y  +384.697, Z    +0.000, E1   +21.693, E3 +577391.772}
SPL {X  -162.820, Y  +382.288, Z    +0.000, E1   +21.742, E3 +577403.895}
SPL {X  -162.817, Y  +379.520, Z    +0.000, E1   +21.723, E3 +577418.733}
SPL {X  -162.776, Y  +376.710, Z    +0.000, E1   +21.698, E3 +577433.472}
SPL {X  -162.707, Y  +374.438, Z    +0.000, E1   +21.688, E3 +577445.476}
SPL {X  -162.607, Y  +372.171, Z    +0.000, E1   +21.692, E3 +577457.275}
SPL {X  -162.494, Y  +370.197, Z    +0.000, E1   +21.655, E3 +577467.902}
SPL {X  -162.349, Y  +368.131, Z    +0.000, E1   +21.624, E3 +577479.020}
SPL {X  -162.161, Y  +365.866, Z    +0.000, E1   +21.642, E3 +577490.705}
SPL {X  -161.651, Y  +361.024, Z    +0.000, E1   +22.970, E3 +577504.128}
SPL {X  -160.281, Y  +351.857, Z    +0.000, E1   +24.243, E3 +577539.467}
ENDSPLINE

SPLINE
SPL {X  -161.833, Y  +362.603, Z    +0.000, E1   +17.021, E3 +577554.163}
ENDSPLINE

SPLINE
SPL {X  -160.786, Y  +354.842, Z    +0.000, E1   +19.274, E3 +577586.319}
ENDSPLINE

SPLINE
SPL {X  -162.485, Y  +370.062, Z    +0.000, E1   +10.606, E3 +577592.697}
SPL {X  -162.818, Y  +379.636, Z    +0.000, E1    +5.115, E3 +577582.046}
SPL {X  -162.820, Y  +386.976, Z    +0.000, E1    +0.144, E3 +577581.145}
SPL {X  -162.820, Y  +390.236, Z    +0.000, E1    -2.204, E3 +577587.203}
SPL {X  -162.820, Y  +393.415, Z    +0.000, E1    -4.587, E3 +577588.487}
SPL {X  -162.820, Y  +399.630, Z    +0.000, E1    -9.426, E3 +577590.417}
SPL {X  -162.820, Y  +408.127, Z    +0.000, E1   -18.417, E3 +577576.705}
SPL {X  -162.820, Y  +420.083, Z    +0.000, E1   -24.325, E3 +577597.181}
SPL {X  -162.820, Y  +428.527, Z    +0.000, E1   -26.988, E3 +577614.473}
SPL {X  -162.820, Y  +431.336, Z    +0.000, E1   -24.162, E3 +577644.683}
SPL {X  -162.820, Y  +432.048, Z    +0.000, E1   -22.832, E3 +577659.187}
SPL {X  -162.820, Y  +434.888, Z    +0.000, E1   -22.823, E3 +577673.136}
SPL {X  -162.820, Y  +436.834, Z    +0.000, E1   -22.779, E3 +577683.096}
SPL {X  -162.820, Y  +438.868, Z    +0.000, E1   -22.837, E3 +577692.750}
SPL {X  -162.820, Y  +441.351, Z    +0.000, E1   -22.805, E3 +577705.325}
SPL {X  -162.820, Y  +443.809, Z    +0.000, E1   -22.804, E3 +577717.491}
SPL {X  -162.820, Y  +446.105, Z    +0.000, E1   -22.815, E3 +577728.734}
SPL {X  -162.820, Y  +447.974, Z    +0.000, E1   -22.856, E3 +577737.637}
SPL {X  -162.820, Y  +449.911, Z    +0.000, E1   -22.774, E3 +577747.911}
SPL {X  -162.820, Y  +451.861, Z    +0.000, E1   -22.750, E3 +577757.759}
SPL {X  -162.820, Y  +454.167, Z    +0.000, E1   -22.842, E3 +577768.488}
SPL {X  -162.820, Y  +456.529, Z    +0.000, E1   -22.855, E3 +577780.017}
SPL {X  -162.820, Y  +458.725, Z    +0.000, E1   -22.793, E3 +577791.421}
SPL {X  -162.820, Y  +461.700, Z    +0.000, E1   -22.822, E3 +577806.044}
SPL {X  -162.820, Y  +464.633, Z    +0.000, E1   -22.813, E3 +577820.540}
SPL {X  -162.820, Y  +466.699, Z    +0.000, E1   -22.824, E3 +577830.587}
SPL {X  -162.820, Y  +468.655, Z    +0.000, E1   -22.858, E3 +577840.030}
SPL {X  -162.820, Y  +470.892, Z    +0.000, E1   -22.837, E3 +577851.269}
SPL {X  -162.820, Y  +473.485, Z    +0.000, E1   -22.806, E3 +577864.467}
SPL {X  -162.820, Y  +476.589, Z    +0.000, E1   -22.788, E3 +577879.989}
SPL {X  -162.820, Y  +478.914, Z    +0.000, E1   -22.821, E3 +577891.087}
SPL {X  -162.820, Y  +481.034, Z    +0.000, E1   -22.831, E3 +577901.609}
SPL {X  -162.820, Y  +484.256, Z    +0.000, E1   -22.840, E3 +577917.628}
SPL {X  -162.820, Y  +487.014, Z    +0.000, E1   -22.789, E3 +577931.495}
SPL {X  -162.820, Y  +489.750, Z    +0.000, E1   -22.832, E3 +577944.869}
SPL {X  -162.820, Y  +493.233, Z    +0.000, E1   -22.844, E3 +577962.006}
SPL {X  -162.820, Y  +496.150, Z    +0.000, E1   -22.796, E3 +577976.726}
SPL {X  -162.820, Y  +498.661, Z    +0.000, E1   -22.828, E3 +577988.907}
SPL {X  -162.820, Y  +501.761, Z    +0.000, E1   -22.820, E3 +578004.475}
SPL {X  -162.820, Y  +505.323, Z    +0.000, E1   -22.838, E3 +578021.922}
SPL {X  -162.820, Y  +507.875, Z    +0.000, E1   -22.849, E3 +578034.289}
SPL {X  -162.820, Y  +510.068, Z    +0.000, E1   -22.761, E3 +578045.982}
SPL {X  -162.820, Y  +512.359, Z    +0.000, E1   -22.823, E3 +578056.714}
SPL {X  -162.820, Y  +514.562, Z    +0.000, E1   -22.806, E3 +578067.901}
SPL {X  -162.820, Y  +517.952, Z    +0.000, E1   -22.864, E3 +578084.298}
SPL {X  -162.820, Y  +520.641, Z    +0.000, E1   -22.790, E3 +578098.017}
SPL {X  -162.820, Y  +522.740, Z    +0.000, E1   -22.811, E3 +578108.259}
SPL {X  -162.820, Y  +524.628, Z    +0.000, E1   -22.846, E3 +578117.254}
SPL {X  -162.820, Y  +526.661, Z    +0.000, E1   -22.801, E3 +578127.810}
SPL {X  -162.820, Y  +529.662, Z    +0.000, E1   -22.810, E3 +578142.660}
SPL {X  -162.820, Y  +532.614, Z    +0.000, E1   -22.828, E3 +578157.067}
SPL {X  -162.820, Y  +534.838, Z    +0.000, E1   -22.864, E3 +578167.695}
SPL {X  -162.820, Y  +536.882, Z    +0.000, E1   -22.782, E3 +578178.550}
SPL {X  -162.820, Y  +539.194, Z    +0.000, E1   -22.826, E3 +578189.599}
SPL {X  -162.820, Y  +541.555, Z    +0.000, E1   -22.817, E3 +578201.413}
SPL {X  -162.820, Y  +543.728, Z    +0.000, E1   -22.799, E3 +578212.271}
SPL {X  -162.820, Y  +545.925, Z    +0.000, E1   -22.803, E3 +578223.141}
SPL {X  -162.820, Y  +548.328, Z    +0.000, E1   -22.796, E3 +578235.136}
SPL {X  -162.820, Y  +551.027, Z    +0.000, E1   -22.819, E3 +578248.329}
SPL {X  -162.820, Y  +553.721, Z    +0.000, E1   -22.807, E3 +578261.773}
SPL {X  -162.820, Y  +556.430, Z    +0.000, E1   -22.821, E3 +578275.069}
SPL {X  -162.820, Y  +559.675, Z    +0.000, E1   -22.837, E3 +578291.149}
SPL {X  -162.820, Y  +562.799, Z    +0.000, E1   -22.814, E3 +578306.655}
SPL {X  -162.820, Y  +565.170, Z    +0.000, E1   -22.801, E3 +578318.480}
SPL {X  -162.820, Y  +568.020, Z    +0.000, E1   -22.787, E3 +578332.867}
SPL {X  -162.820, Y  +570.992, Z    +0.000, E1   -22.834, E3 +578347.086}
SPL {X  -162.820, Y  +572.901, Z    +0.000, E1   -22.775, E3 +578356.955}
SPL {X  -162.820, Y  +575.638, Z    +0.000, E1   -22.855, E3 +578370.064}
SPL {X  -162.820, Y  +578.553, Z    +0.000, E1   -22.801, E3 +578384.776}
SPL {X  -162.820, Y  +581.064, Z    +0.000, E1   -22.823, E3 +578397.061}
SPL {X  -162.820, Y  +583.435, Z    +0.000, E1   -22.808, E3 +578408.883}
SPL {X  -162.820, Y  +585.410, Z    +0.000, E1   -22.764, E3 +578419.018}
SPL {X  -162.820, Y  +587.676, Z    +0.000, E1   -22.853, E3 +578429.533}
SPL {X  -162.820, Y  +589.682, Z    +0.000, E1   -22.776, E3 +578440.063}
SPL {X  -162.820, Y  +591.720, Z    +0.000, E1   -22.868, E3 +578449.374}
SPL {X  -162.820, Y  +593.650, Z    +0.000, E1   -22.810, E3 +578459.443}
SPL {X  -162.820, Y  +595.830, Z    +0.000, E1   -22.828, E3 +578470.059}
SPL {X  -162.820, Y  +598.094, Z    +0.000, E1   -22.843, E3 +578481.172}
SPL {X  -162.820, Y  +600.420, Z    +0.000, E1   -22.826, E3 +578492.804}
SPL {X  -162.820, Y  +602.573, Z    +0.000, E1   -22.830, E3 +578503.389}
SPL {X  -162.820, Y  +604.828, Z    +0.000, E1   -22.784, E3 +578515.027}
SPL {X  -162.820, Y  +607.142, Z    +0.000, E1   -22.808, E3 +578526.208}
SPL {X  -162.820, Y  +608.890, Z    +0.000, E1   -22.790, E3 +578535.032}
SPL {X  -162.820, Y  +611.103, Z    +0.000, E1   -22.785, E3 +578546.071}
SPL {X  -162.820, Y  +613.294, Z    +0.000, E1   -22.780, E3 +578556.944}
SPL {X  -162.820, Y  +615.356, Z    +0.000, E1   -22.799, E3 +578567.001}
SPL {X  -162.820, Y  +617.439, Z    +0.000, E1   -22.808, E3 +578577.259}
SPL {X  -162.820, Y  +619.665, Z    +0.000, E1   -22.817, E3 +578588.227}
SPL {X  -162.820, Y  +621.733, Z    +0.000, E1   -22.759, E3 +578598.951}
SPL {X  -162.820, Y  +624.076, Z    +0.000, E1   -22.774, E3 +578610.456}
SPL {X  -162.820, Y  +627.244, Z    +0.000, E1   -22.803, E3 +578626.139}
SPL {X  -162.820, Y  +630.349, Z    +0.000, E1   -22.766, E3 +578641.671}
SPL {X  -162.820, Y  +632.572, Z    +0.000, E1   -22.785, E3 +578652.477}
SPL {X  -162.820, Y  +634.507, Z    +0.000, E1   -22.784, E3 +578662.116}
SPL {X  -162.820, Y  +636.863, Z    +0.000, E1   -22.760, E3 +578674.038}
SPL {X  -162.820, Y  +639.254, Z    +0.000, E1   -22.767, E3 +578685.822}
SPL {X  -162.820, Y  +641.195, Z    +0.000, E1   -22.782, E3 +578695.269}
SPL {X  -162.820, Y  +643.449, Z    +0.000, E1   -22.796, E3 +578706.439}
SPL {X  -162.820, Y  +645.630, Z    +0.000, E1   -22.795, E3 +578717.135}
SPL {X  -162.820, Y  +647.561, Z    +0.000, E1   -22.705, E3 +578727.586}
SPL {X  -162.820, Y  +651.051, Z    +0.000, E1   -22.833, E3 +578744.005}
SPL {X  -162.820, Y  +653.898, Z    +0.000, E1   -22.796, E3 +578758.191}
SPL {X  -162.820, Y  +656.161, Z    +0.000, E1   -22.812, E3 +578769.312}
SPL {X  -162.820, Y  +658.384, Z    +0.000, E1   -22.822, E3 +578780.179}
SPL {X  -162.820, Y  +660.215, Z    +0.000, E1   -22.649, E3 +578790.769}
SPL {X  -162.820, Y  +662.823, Z    +0.000, E1   -22.799, E3 +578802.477}
SPL {X  -162.820, Y  +665.112, Z    +0.000, E1   -22.835, E3 +578813.532}
SPL {X  -162.820, Y  +667.016, Z    +0.000, E1   -22.823, E3 +578822.960}
SPL {X  -162.820, Y  +668.960, Z    +0.000, E1   -22.773, E3 +578833.127}
SPL {X  -162.820, Y  +672.333, Z    +0.000, E1   -22.837, E3 +578849.463}
SPL {X  -162.812, Y  +675.071, Z    +0.000, E1   -22.742, E3 +578863.609}
SPL {X  -162.773, Y  +677.428, Z    +0.000, E1   -22.762, E3 +578875.206}
SPL {X  -162.691, Y  +679.987, Z    +0.000, E1   -22.794, E3 +578887.619}
SPL {X  -162.559, Y  +682.717, Z    +0.000, E1   -22.726, E3 +578901.803}
SPL {X  -162.404, Y  +685.137, Z    +0.000, E1   -22.766, E3 +578913.325}
SPL {X  -162.229, Y  +687.364, Z    +0.000, E1   -22.685, E3 +578925.194}
SPL {X  -161.938, Y  +690.422, Z    +0.000, E1   -22.769, E3 +578939.600}
SPL {X  -161.065, Y  +697.344, Z    +0.000, E1   -25.698, E3 +578948.719}
SPL {X  -158.730, Y  +709.763, Z    +0.000, E1   -31.225, E3 +578957.393}
ENDSPLINE

SPLINE
SPL {X  -160.932, Y  +698.225, Z    +0.000, E1   -21.712, E3 +578988.502}
SPL {X  -161.691, Y  +692.643, Z    +0.000, E1   -17.369, E3 +579005.385}
SPL {X  -162.534, Y  +683.153, Z    +0.000, E1   -10.475, E3 +579030.852}
SPL {X  -162.820, Y  +670.105, Z    +0.000, E1    -2.484, E3 +579023.499}
SPL {X  -162.820, Y  +665.819, Z    +0.000, E1    +0.492, E3 +579025.795}
SPL {X  -162.820, Y  +661.883, Z    +0.000, E1    +3.373, E3 +579030.271}
SPL {X  -162.820, Y  +655.163, Z    +0.000, E1    +8.702, E3 +579029.870}
SPL {X  -162.820, Y  +634.515, Z    +0.000, E1   +26.439, E3 +579022.283}
ENDSPLINE

SPLINE
SPL {X  -162.820, Y  +638.080, Z    +0.000, E1   +18.858, E3 +579052.248}
ENDSPLINE

SPLINE
SPL {X  -162.820, Y  +623.278, Z    +0.000, E1   +28.723, E3 +579053.818}
SPL {X  -162.820, Y  +618.658, Z    +0.000, E1   +26.841, E3 +579082.427}
ENDSPLINE

SPLINE
SPL {X  -162.820, Y  +623.685, Z    +0.000, E1   +22.346, E3 +579094.734}
ENDSPLINE

SPLINE
SPL {X  -162.820, Y  +621.304, Z    +0.000, E1   +22.259, E3 +579107.549}
SPL {X  -162.820, Y  +618.758, Z    +0.000, E1   +22.239, E3 +579120.700}
SPL {X  -162.820, Y  +616.062, Z    +0.000, E1   +22.275, E3 +579134.120}
SPL {X  -162.820, Y  +613.536, Z    +0.000, E1   +22.242, E3 +579147.242}
SPL {X  -162.820, Y  +611.128, Z    +0.000, E1   +22.252, E3 +579159.413}
SPL {X  -162.820, Y  +608.428, Z    +0.000, E1   +22.255, E3 +579173.196}
SPL {X  -162.820, Y  +605.984, Z    +0.000, E1   +22.221, E3 +579185.833}
SPL {X  -162.820, Y  +603.020, Z    +0.000, E1   +22.272, E3 +579200.731}
SPL {X  -162.820, Y  +599.842, Z    +0.000, E1   +22.298, E3 +579216.497}
SPL {X  -162.820, Y  +597.194, Z    +0.000, E1   +22.253, E3 +579230.418}
SPL {X  -162.820, Y  +594.779, Z    +0.000, E1   +22.284, E3 +579242.322}
SPL {X  -162.820, Y  +592.389, Z    +0.000, E1   +22.245, E3 +579254.938}
SPL {X  -162.820, Y  +589.492, Z    +0.000, E1   +22.304, E3 +579269.123}
SPL {X  -162.820, Y  +587.447, Z    +0.000, E1   +22.279, E3 +579279.652}
SPL {X  -162.820, Y  +585.192, Z    +0.000, E1   +22.298, E3 +579291.062}
SPL {X  -162.820, Y  +582.610, Z    +0.000, E1   +22.234, E3 +579304.685}
SPL {X  -162.820, Y  +579.691, Z    +0.000, E1   +22.312, E3 +579318.957}
SPL {X  -162.820, Y  +577.460, Z    +0.000, E1   +22.218, E3 +579330.944}
SPL {X  -162.820, Y  +575.394, Z    +0.000, E1   +22.240, E3 +579341.369}
SPL {X  -162.820, Y  +572.645, Z    +0.000, E1   +22.246, E3 +579355.366}
SPL {X  -162.820, Y  +570.282, Z    +0.000, E1   +22.231, E3 +579367.417}
SPL {X  -162.820, Y  +567.961, Z    +0.000, E1   +22.247, E3 +579379.206}
SPL {X  -162.820, Y  +564.506, Z    +0.000, E1   +22.298, E3 +579396.520}
SPL {X  -162.820, Y  +561.620, Z    +0.000, E1   +22.191, E3 +579411.901}
SPL {X  -162.820, Y  +559.515, Z    +0.000, E1   +22.273, E3 +579421.903}
SPL {X  -162.820, Y  +556.723, Z    +0.000, E1   +22.309, E3 +579435.987}
SPL {X  -162.820, Y  +554.378, Z    +0.000, E1   +22.288, E3 +579447.832}
SPL {X  -162.820, Y  +552.787, Z    +0.000, E1   +22.213, E3 +579456.654}
SPL {X  -162.820, Y  +550.871, Z    +0.000, E1   +22.229, E3 +579466.249}
SPL {X  -162.820, Y  +548.168, Z    +0.000, E1   +22.298, E3 +579479.585}
SPL {X  -162.820, Y  +545.860, Z    +0.000, E1   +22.216, E3 +579491.843}
SPL {X  -162.820, Y  +543.558, Z    +0.000, E1   +22.285, E3 +579503.073}
SPL {X  -162.820, Y  +540.968, Z    +0.000, E1   +22.274, E3 +579516.345}
SPL {X  -162.820, Y  +538.512, Z    +0.000, E1   +22.287, E3 +579528.658}
SPL {X  -162.820, Y  +535.523, Z    +0.000, E1   +22.266, E3 +579544.273}
SPL {X  -162.820, Y  +531.757, Z    +0.000, E1   +22.276, E3 +579563.328}
SPL {X  -162.820, Y  +527.980, Z    +0.000, E1   +22.326, E3 +579582.159}
SPL {X  -162.820, Y  +524.599, Z    +0.000, E1   +22.287, E3 +579599.556}
SPL {X  -162.820, Y  +522.011, Z    +0.000, E1   +22.282, E3 +579612.633}
SPL {X  -162.820, Y  +519.457, Z    +0.000, E1   +22.481, E3 +579623.922}
SPL {X  -162.820, Y  +505.859, Z    +0.000, E1   +28.367, E3 +579638.405}
SPL {X  -162.820, Y  +504.131, Z    +0.000, E1   +27.325, E3 +579652.544}
SPL {X  -162.820, Y  +502.813, Z    +0.000, E1   +26.013, E3 +579667.920}
SPL {X  -162.820, Y  +502.016, Z    +0.000, E1   +24.802, E3 +579680.263}
SPL {X  -162.820, Y  +501.060, Z    +0.000, E1   +24.081, E3 +579690.452}
SPL {X  -162.820, Y  +499.934, Z    +0.000, E1   +22.814, E3 +579706.321}
SPL {X  -162.820, Y  +498.303, Z    +0.000, E1   +21.749, E3 +579723.577}
SPL {X  -162.820, Y  +495.897, Z    +0.000, E1   +21.662, E3 +579736.731}
SPL {X  -162.820, Y  +493.717, Z    +0.000, E1   +21.704, E3 +579747.837}
SPL {X  -162.820, Y  +491.396, Z    +0.000, E1   +21.707, E3 +579759.961}
SPL {X  -162.820, Y  +489.485, Z    +0.000, E1   +21.661, E3 +579770.309}
SPL {X  -162.820, Y  +487.723, Z    +0.000, E1   +21.665, E3 +579779.512}
SPL {X  -162.820, Y  +485.661, Z    +0.000, E1   +21.712, E3 +579789.956}
SPL {X  -162.820, Y  +482.775, Z    +0.000, E1   +21.716, E3 +579805.208}
SPL {X  -162.820, Y  +479.894, Z    +0.000, E1   +21.695, E3 +579820.284}
SPL {X  -162.820, Y  +477.685, Z    +0.000, E1   +21.656, E3 +579832.222}
SPL {X  -162.820, Y  +475.419, Z    +0.000, E1   +21.711, E3 +579843.575}
SPL {X  -162.820, Y  +473.301, Z    +0.000, E1   +21.712, E3 +579854.672}
SPL {X  -162.820, Y  +470.965, Z    +0.000, E1   +21.700, E3 +579867.017}
SPL {X  -162.820, Y  +469.036, Z    +0.000, E1   +21.695, E3 +579877.060}
SPL {X  -162.820, Y  +467.138, Z    +0.000, E1   +21.678, E3 +579887.232}
SPL {X  -162.820, Y  +465.011, Z    +0.000, E1   +21.692, E3 +579898.215}
SPL {X  -162.820, Y  +462.669, Z    +0.000, E1   +21.752, E3 +579909.995}
SPL {X  -162.820, Y  +460.725, Z    +0.000, E1   +21.689, E3 +579920.608}
SPL {X  -162.820, Y  +458.666, Z    +0.000, E1   +21.695, E3 +579931.420}
SPL {X  -162.820, Y  +456.431, Z    +0.000, E1   +21.708, E3 +579942.949}
SPL {X  -162.820, Y  +453.609, Z    +0.000, E1   +21.757, E3 +579957.483}
SPL {X  -162.820, Y  +450.610, Z    +0.000, E1   +21.698, E3 +579973.540}
SPL {X  -162.820, Y  +448.170, Z    +0.000, E1   +21.667, E3 +579986.561}
SPL {X  -162.820, Y  +446.246, Z    +0.000, E1   +21.696, E3 +579996.378}
SPL {X  -162.820, Y  +443.784, Z    +0.000, E1   +21.713, E3 +580009.165}
SPL {X  -162.820, Y  +440.567, Z    +0.000, E1   +21.731, E3 +580026.004}
SPL {X  -162.820, Y  +437.628, Z    +0.000, E1   +21.678, E3 +580041.668}
SPL {X  -162.820, Y  +435.262, Z    +0.000, E1   +21.727, E3 +580053.604}
SPL {X  -162.820, Y  +433.510, Z    +0.000, E1   +21.692, E3 +580063.018}
SPL {X  -162.820, Y  +431.492, Z    +0.000, E1   +21.686, E3 +580073.713}
SPL {X  -162.820, Y  +429.074, Z    +0.000, E1   +21.710, E3 +580086.165}
SPL {X  -162.820, Y  +427.020, Z    +0.000, E1   +21.674, E3 +580097.167}
SPL {X  -162.820, Y  +424.525, Z    +0.000, E1   +21.712, E3 +580110.080}
SPL {X  -162.820, Y  +421.144, Z    +0.000, E1   +21.719, E3 +580127.747}
SPL {X  -162.820, Y  +418.116, Z    +0.000, E1   +21.761, E3 +580143.078}
SPL {X  -162.820, Y  +416.127, Z    +0.000, E1   +21.715, E3 +580153.783}
SPL {X  -162.820, Y  +414.361, Z    +0.000, E1   +21.613, E3 +580163.970}
SPL {X  -162.820, Y  +412.134, Z    +0.000, E1   +21.697, E3 +580174.915}
SPL {X  -162.820, Y  +409.248, Z    +0.000, E1   +21.741, E3 +580189.850}
SPL {X  -162.820, Y  +406.238, Z    +0.000, E1   +21.697, E3 +580205.818}
SPL {X  -162.820, Y  +404.001, Z    +0.000, E1   +21.723, E3 +580217.248}
SPL {X  -162.820, Y  +402.223, Z    +0.000, E1   +21.697, E3 +580226.733}
SPL {X  -162.820, Y  +400.348, Z    +0.000, E1   +21.713, E3 +580236.459}
SPL {X  -162.820, Y  +398.298, Z    +0.000, E1   +21.721, E3 +580247.074}
SPL {X  -162.820, Y  +396.371, Z    +0.000, E1   +21.713, E3 +580257.256}
SPL {X  -162.820, Y  +394.508, Z    +0.000, E1   +21.616, E3 +580267.812}
SPL {X  -162.820, Y  +392.435, Z    +0.000, E1   +21.681, E3 +580278.165}
SPL {X  -162.820, Y  +389.390, Z    +0.000, E1   +21.742, E3 +580293.772}
SPL {X  -162.820, Y  +386.818, Z    +0.000, E1   +21.679, E3 +580307.531}
SPL {X  -162.820, Y  +384.697, Z    +0.000, E1   +21.693, E3 +580318.601}
SPL {X  -162.820, Y  +382.288, Z    +0.000, E1   +21.742, E3 +580330.725}
SPL {X  -162.820, Y  +380.381, Z    +0.000, E1   +21.655, E3 +580341.450}
SPL {X  -162.808, Y  +378.512, Z    +0.000, E1   +21.736, E3 +580350.502}
SPL {X  -162.776, Y  +376.710, Z    +0.000, E1   +21.698, E3 +580360.301}
SPL {X  -162.707, Y  +374.438, Z    +0.000, E1   +21.688, E3 +580372.305}
SPL {X  -162.607, Y  +372.171, Z    +0.000, E1   +21.692, E3 +580384.105}
SPL {X  -162.494, Y  +370.197, Z    +0.000, E1   +21.655, E3 +580394.731}
SPL {X  -162.349, Y  +368.131, Z    +0.000, E1   +21.624, E3 +580405.849}
SPL {X  -162.161, Y  +365.866, Z    +0.000, E1   +21.642, E3 +580417.534}
SPL {X  -161.927, Y  +363.466, Z    +0.000, E1   +21.730, E3 +580429.306}
SPL {X  -160.290, Y  +351.907, Z    +0.000, E1   +27.562, E3 +580436.883}
SPL {X  -159.725, Y  +348.905, Z    +0.000, E1   +26.136, E3 +580462.118}
ENDSPLINE

SPLINE
SPL {X  -160.871, Y  +355.385, Z    +0.000, E1   +21.841, E3 +580470.961}
SPL {X  -161.833, Y  +362.603, Z    +0.000, E1   +17.021, E3 +580480.992}
ENDSPLINE

SPLINE
SPL {X  -160.786, Y  +354.842, Z    +0.000, E1   +19.274, E3 +580513.148}
ENDSPLINE

SPLINE
SPL {X  -162.485, Y  +370.062, Z    +0.000, E1   +10.606, E3 +580519.526}
SPL {X  -162.818, Y  +379.636, Z    +0.000, E1    +5.115, E3 +580508.875}
SPL {X  -162.820, Y  +386.976, Z    +0.000, E1    +0.144, E3 +580507.974}
SPL {X  -162.820, Y  +391.982, Z    +0.000, E1    -3.443, E3 +580514.739}
SPL {X  -162.820, Y  +399.630, Z    +0.000, E1    -9.426, E3 +580517.246}
SPL {X  -162.820, Y  +408.127, Z    +0.000, E1   -18.417, E3 +580503.535}
SPL {X  -162.820, Y  +420.083, Z    +0.000, E1   -24.325, E3 +580524.010}
SPL {X  -162.820, Y  +428.527, Z    +0.000, E1   -26.988, E3 +580541.302}
SPL {X  -162.820, Y  +431.336, Z    +0.000, E1   -24.162, E3 +580571.512}
SPL {X  -162.820, Y  +432.048, Z    +0.000, E1   -22.832, E3 +580586.016}
SPL {X  -162.820, Y  +434.888, Z    +0.000, E1   -22.823, E3 +580599.966}
SPL {X  -162.820, Y  +436.834, Z    +0.000, E1   -22.779, E3 +580609.926}
SPL {X  -162.820, Y  +438.868, Z    +0.000, E1   -22.837, E3 +580619.579}
SPL {X  -162.820, Y  +441.351, Z    +0.000, E1   -22.805, E3 +580632.154}
SPL {X  -162.820, Y  +443.809, Z    +0.000, E1   -22.804, E3 +580644.321}
SPL {X  -162.820, Y  +446.105, Z    +0.000, E1   -22.815, E3 +580655.563}
SPL {X  -162.820, Y  +447.974, Z    +0.000, E1   -22.856, E3 +580664.466}
SPL {X  -162.820, Y  +449.911, Z    +0.000, E1   -22.774, E3 +580674.741}
SPL {X  -162.820, Y  +451.861, Z    +0.000, E1   -22.750, E3 +580684.588}
SPL {X  -162.820, Y  +454.167, Z    +0.000, E1   -22.842, E3 +580695.318}
SPL {X  -162.820, Y  +456.529, Z    +0.000, E1   -22.855, E3 +580706.846}
SPL {X  -162.820, Y  +458.725, Z    +0.000, E1   -22.793, E3 +580718.250}
SPL {X  -162.820, Y  +461.700, Z    +0.000, E1   -22.822, E3 +580732.873}
SPL {X  -162.820, Y  +464.633, Z    +0.000, E1   -22.813, E3 +580747.370}
SPL {X  -162.820, Y  +466.699, Z    +0.000, E1   -22.824, E3 +580757.416}
SPL {X  -162.820, Y  +468.655, Z    +0.000, E1   -22.858, E3 +580766.859}
SPL {X  -162.820, Y  +470.892, Z    +0.000, E1   -22.837, E3 +580778.098}
SPL {X  -162.820, Y  +472.726, Z    +0.000, E1   -22.777, E3 +580787.637}
SPL {X  -162.820, Y  +475.118, Z    +0.000, E1   -22.777, E3 +580799.608}
SPL {X  -162.820, Y  +478.177, Z    +0.000, E1   -22.834, E3 +580814.301}
SPL {X  -162.820, Y  +481.034, Z    +0.000, E1   -22.831, E3 +580828.439}
SPL {X  -162.820, Y  +483.391, Z    +0.000, E1   -22.793, E3 +580840.375}
SPL {X  -162.820, Y  +486.307, Z    +0.000, E1   -22.833, E3 +580854.629}
SPL {X  -162.820, Y  +488.828, Z    +0.000, E1   -22.793, E3 +580867.271}
SPL {X  -162.820, Y  +491.768, Z    +0.000, E1   -22.852, E3 +580881.568}
SPL {X  -162.820, Y  +495.526, Z    +0.000, E1   -22.833, E3 +580900.340}
SPL {X  -162.820, Y  +499.330, Z    +0.000, E1   -22.841, E3 +580919.121}
SPL {X  -162.820, Y  +503.049, Z    +0.000, E1   -22.823, E3 +580937.670}
SPL {X  -162.820, Y  +505.970, Z    +0.000, E1   -22.835, E3 +580951.843}
SPL {X  -162.820, Y  +508.611, Z    +0.000, E1   -22.838, E3 +580965.014}
SPL {X  -162.820, Y  +511.620, Z    +0.000, E1   -22.791, E3 +580980.258}
SPL {X  -162.820, Y  +513.873, Z    +0.000, E1   -22.800, E3 +580991.230}
SPL {X  -162.820, Y  +516.100, Z    +0.000, E1   -22.809, E3 +581002.306}
SPL {X  -162.820, Y  +518.662, Z    +0.000, E1   -22.847, E3 +581014.605}
SPL {X  -162.820, Y  +520.641, Z    +0.000, E1   -22.790, E3 +581024.846}
SPL {X  -162.820, Y  +522.740, Z    +0.000, E1   -22.811, E3 +581035.088}
SPL {X  -162.820, Y  +525.255, Z    +0.000, E1   -22.822, E3 +581047.509}
SPL {X  -162.820, Y  +528.050, Z    +0.000, E1   -22.808, E3 +581061.473}
SPL {X  -162.820, Y  +530.303, Z    +0.000, E1   -22.798, E3 +581072.627}
SPL {X  -162.820, Y  +532.614, Z    +0.000, E1   -22.828, E3 +581083.896}
SPL {X  -162.820, Y  +534.838, Z    +0.000, E1   -22.864, E3 +581094.525}
SPL {X  -162.820, Y  +536.882, Z    +0.000, E1   -22.782, E3 +581105.380}
SPL {X  -162.820, Y  +539.194, Z    +0.000, E1   -22.826, E3 +581116.428}
SPL {X  -162.820, Y  +541.555, Z    +0.000, E1   -22.817, E3 +581128.242}
SPL {X  -162.820, Y  +543.728, Z    +0.000, E1   -22.799, E3 +581139.100}
SPL {X  -162.820, Y  +545.925, Z    +0.000, E1   -22.803, E3 +581149.970}
SPL {X  -162.820, Y  +549.071, Z    +0.000, E1   -22.836, E3 +581165.497}
SPL {X  -162.820, Y  +553.089, Z    +0.000, E1   -22.838, E3 +581185.397}
SPL {X  -162.820, Y  +556.430, Z    +0.000, E1   -22.821, E3 +581201.898}
SPL {X  -162.820, Y  +558.974, Z    +0.000, E1   -22.806, E3 +581214.598}
SPL {X  -162.820, Y  +562.171, Z    +0.000, E1   -22.845, E3 +581230.296}
SPL {X  -162.820, Y  +565.170, Z    +0.000, E1   -22.801, E3 +581245.310}
SPL {X  -162.820, Y  +567.308, Z    +0.000, E1   -22.750, E3 +581256.326}
SPL {X  -162.820, Y  +570.378, Z    +0.000, E1   -22.843, E3 +581270.950}
SPL {X  -162.820, Y  +573.634, Z    +0.000, E1   -22.827, E3 +581287.094}
SPL {X  -162.820, Y  +576.228, Z    +0.000, E1   -22.814, E3 +581299.990}
SPL {X  -162.820, Y  +578.553, Z    +0.000, E1   -22.801, E3 +581311.606}
SPL {X  -162.820, Y  +581.064, Z    +0.000, E1   -22.823, E3 +581323.890}
SPL {X  -162.820, Y  +583.435, Z    +0.000, E1   -22.808, E3 +581335.712}
SPL {X  -162.820, Y  +585.410, Z    +0.000, E1   -22.764, E3 +581345.848}
SPL {X  -162.820, Y  +587.676, Z    +0.000, E1   -22.853, E3 +581356.362}
SPL {X  -162.820, Y  +589.682, Z    +0.000, E1   -22.776, E3 +581366.892}
SPL {X  -162.820, Y  +591.720, Z    +0.000, E1   -22.868, E3 +581376.203}
SPL {X  -162.820, Y  +593.650, Z    +0.000, E1   -22.810, E3 +581386.273}
SPL {X  -162.820, Y  +595.830, Z    +0.000, E1   -22.828, E3 +581396.889}
SPL {X  -162.820, Y  +598.094, Z    +0.000, E1   -22.843, E3 +581408.002}
SPL {X  -162.820, Y  +600.420, Z    +0.000, E1   -22.826, E3 +581419.633}
SPL {X  -162.820, Y  +602.573, Z    +0.000, E1   -22.830, E3 +581430.218}
SPL {X  -162.820, Y  +604.828, Z    +0.000, E1   -22.784, E3 +581441.856}
SPL {X  -162.820, Y  +607.142, Z    +0.000, E1   -22.808, E3 +581453.037}
SPL {X  -162.820, Y  +608.890, Z    +0.000, E1   -22.790, E3 +581461.862}
SPL {X  -162.820, Y  +611.103, Z    +0.000, E1   -22.785, E3 +581472.900}
SPL {X  -162.820, Y  +613.294, Z    +0.000, E1   -22.780, E3 +581483.773}
SPL {X  -162.820, Y  +615.356, Z    +0.000, E1   -22.799, E3 +581493.830}
SPL {X  -162.820, Y  +617.439, Z    +0.000, E1   -22.808, E3 +581504.088}
SPL {X  -162.820, Y  +619.665, Z    +0.000, E1   -22.817, E3 +581515.056}
SPL {X  -162.820, Y  +621.733, Z    +0.000, E1   -22.759, E3 +581525.781}
SPL {X  -162.820, Y  +624.076, Z    +0.000, E1   -22.774, E3 +581537.286}
SPL {X  -162.820, Y  +626.527, Z    +0.000, E1   -22.768, E3 +581549.528}
SPL {X  -162.820, Y  +629.758, Z    +0.000, E1   -22.800, E3 +581565.457}
SPL {X  -162.820, Y  +632.572, Z    +0.000, E1   -22.785, E3 +581579.307}
SPL {X  -162.820, Y  +634.507, Z    +0.000, E1   -22.784, E3 +581588.945}
SPL {X  -162.820, Y  +636.863, Z    +0.000, E1   -22.760, E3 +581600.868}
SPL {X  -162.820, Y  +639.254, Z    +0.000, E1   -22.767, E3 +581612.651}
SPL {X  -162.820, Y  +641.195, Z    +0.000, E1   -22.782, E3 +581622.098}
SPL {X  -162.820, Y  +643.449, Z    +0.000, E1   -22.796, E3 +581633.268}
SPL {X  -162.820, Y  +645.630, Z    +0.000, E1   -22.795, E3 +581643.964}
SPL {X  -162.820, Y  +647.561, Z    +0.000, E1   -22.705, E3 +581654.415}
SPL {X  -162.820, Y  +651.051, Z    +0.000, E1   -22.833, E3 +581670.834}
SPL {X  -162.820, Y  +653.898, Z    +0.000, E1   -22.796, E3 +581685.020}
SPL {X  -162.820, Y  +656.161, Z    +0.000, E1   -22.812, E3 +581696.142}
SPL {X  -162.820, Y  +658.384, Z    +0.000, E1   -22.822, E3 +581707.008}
SPL {X  -162.820, Y  +660.215, Z    +0.000, E1   -22.649, E3 +581717.598}
SPL {X  -162.820, Y  +662.823, Z    +0.000, E1   -22.799, E3 +581729.306}
SPL {X  -162.820, Y  +665.112, Z    +0.000, E1   -22.835, E3 +581740.361}
SPL {X  -162.820, Y  +667.016, Z    +0.000, E1   -22.823, E3 +581749.789}
SPL {X  -162.820, Y  +668.960, Z    +0.000, E1   -22.773, E3 +581759.957}
SPL {X  -162.820, Y  +672.333, Z    +0.000, E1   -22.837, E3 +581776.293}
SPL {X  -162.812, Y  +675.071, Z    +0.000, E1   -22.742, E3 +581790.438}
SPL {X  -162.773, Y  +677.428, Z    +0.000, E1   -22.762, E3 +581802.035}
SPL {X  -162.691, Y  +679.987, Z    +0.000, E1   -22.794, E3 +581814.449}
SPL {X  -162.604, Y  +681.880, Z    +0.000, E1   -22.691, E3 +581824.609}
SPL {X  -162.458, Y  +684.346, Z    +0.000, E1   -22.764, E3 +581836.403}
SPL {X  -162.296, Y  +686.547, Z    +0.000, E1   -22.660, E3 +581848.020}
SPL {X  -162.090, Y  +688.902, Z    +0.000, E1   -22.700, E3 +581859.528}
SPL {X  -161.474, Y  +694.390, Z    +0.000, E1   -24.298, E3 +581872.883}
SPL {X  -158.730, Y  +709.763, Z    +0.000, E1   -31.225, E3 +581884.222}
ENDSPLINE

SPLINE
SPL {X  -160.932, Y  +698.225, Z    +0.000, E1   -21.712, E3 +581915.331}
SPL {X  -161.917, Y  +690.622, Z    +0.000, E1   -16.445, E3 +581928.932}
ENDSPLINE

SPLINE
SPL {X  -161.349, Y  +695.340, Z    +0.000, E1   -18.625, E3 +581936.550}
ENDSPLINE

SPLINE
SPL {X  -162.534, Y  +683.153, Z    +0.000, E1   -10.475, E3 +581957.681}
SPL {X  -162.820, Y  +667.630, Z    +0.000, E1    -0.882, E3 +581951.657}
SPL {X  -162.820, Y  +661.883, Z    +0.000, E1    +3.373, E3 +581957.101}
SPL {X  -162.820, Y  +653.808, Z    +0.000, E1    +9.891, E3 +581954.792}
SPL {X  -162.820, Y  +632.548, Z    +0.000, E1   +27.446, E3 +581951.329}
ENDSPLINE

SPLINE
SPL {X  -162.820, Y  +638.080, Z    +0.000, E1   +18.858, E3 +581979.077}
ENDSPLINE

SPLINE
SPL {X  -162.820, Y  +623.278, Z    +0.000, E1   +28.723, E3 +581980.648}
SPL {X  -162.820, Y  +618.658, Z    +0.000, E1   +26.841, E3 +582009.257}
ENDSPLINE

SPLINE
SPL {X  -162.820, Y  +623.685, Z    +0.000, E1   +22.346, E3 +582021.563}
ENDSPLINE

